TYPE "typeSmcChillerHrle90a40cmIo"
// stored: IsFailsafeCompliant false
   STRUCT
      in { ExternalAccessible := 'False'; ExternalVisible := 'False'; ExternalWritable := 'False'} : Struct   // Lesen / Read
         fluidDischargeTempCH1 { ExternalAccessible := 'False'; ExternalVisible := 'False'; ExternalWritable := 'False'} : Real;   // Austrittstemperatur der zirkulierenden Flüssigkeit Kanal 1 / Outlet temperature of the circulating fluid channel 1
         fluidDischargeTempCH2 { ExternalAccessible := 'False'; ExternalVisible := 'False'; ExternalWritable := 'False'} : Real;   // Austrittstemperatur der zirkulierenden Flüssigkeit Kanal 2 / Outlet temperature of the circulating fluid channel 2
         reserve1 { ExternalAccessible := 'False'; ExternalVisible := 'False'; ExternalWritable := 'False'} : Word;   // Reserve
         reserve2 { ExternalAccessible := 'False'; ExternalVisible := 'False'; ExternalWritable := 'False'} : Word;   // Reserve
         fluidDischargePressureCH1 { ExternalAccessible := 'False'; ExternalVisible := 'False'; ExternalWritable := 'False'} : Real;   // Förderdruck der zirkulierenden Flüssigkeit Kanal 1 / Delivery pressure of the circulating fluid channel 1
         reserve3 { ExternalAccessible := 'False'; ExternalVisible := 'False'; ExternalWritable := 'False'} : Word;   // Reserve
         reserve4 { ExternalAccessible := 'False'; ExternalVisible := 'False'; ExternalWritable := 'False'} : Word;   // Reserve
         reserve5 { ExternalAccessible := 'False'; ExternalVisible := 'False'; ExternalWritable := 'False'} : Word;   // Reserve
         dataDisplay1 { ExternalAccessible := 'False'; ExternalVisible := 'False'; ExternalWritable := 'False'} : Real;   // Datenanzeige 1 / Data display 1
         dataDisplay2 { ExternalAccessible := 'False'; ExternalVisible := 'False'; ExternalWritable := 'False'} : Real;   // Datenanzeige 2 / Data display 2
         statusFlags1 { ExternalAccessible := 'False'; ExternalVisible := 'False'; ExternalWritable := 'False'} : Array[0..15] of Bool;   // Statuskennzeichen 1 / Status identifier 1
         alarmFlags1 { ExternalAccessible := 'False'; ExternalVisible := 'False'; ExternalWritable := 'False'} : Array[0..15] of Bool;   // Alarmmerker 1 / Alarm flag 1
         alarmFlags2 { ExternalAccessible := 'False'; ExternalVisible := 'False'; ExternalWritable := 'False'} : Array[0..15] of Bool;   // Alarmmerker 2 / Alarm flag 2
         alarmFlags3 { ExternalAccessible := 'False'; ExternalVisible := 'False'; ExternalWritable := 'False'} : Array[0..15] of Bool;   // Alarmmerker 3 / Alarm flag 3
         alarmFlags4 { ExternalAccessible := 'False'; ExternalVisible := 'False'; ExternalWritable := 'False'} : Array[0..15] of Bool;   // Alarmmerker 4 / Alarm flag 4
         alarmFlags5 { ExternalAccessible := 'False'; ExternalVisible := 'False'; ExternalWritable := 'False'} : Array[0..15] of Bool;   // Alarmmerker 5 / Alarm flag 5
      END_STRUCT;
      inOut { ExternalAccessible := 'False'; ExternalVisible := 'False'; ExternalWritable := 'False'} : Struct   // Lesen/Schreiben / Read/write
         fluidSetTempCH1 { ExternalAccessible := 'False'; ExternalVisible := 'False'; ExternalWritable := 'False'} : Real;   // Solltemperatur der zirkulierenden Flüssigkeit / Target temperature of the circulating fluid
         fluidSetTempCH2 { ExternalAccessible := 'False'; ExternalVisible := 'False'; ExternalWritable := 'False'} : Real;   // Umwälzflüssigkeitssolltemperatur als Offset von Kanal 1 (Sollwert Kanal 2 = Sollwert Kanal 1 + Offset Kanal 2) / Circulating fluid target temperature as offset for channel 1 (target value channel 2 = target value channel 1 + offset channel 2)
         controlBits { ExternalAccessible := 'False'; ExternalVisible := 'False'; ExternalWritable := 'False'} : Array[0..15] of Bool;   // Steuerbits / Control bits
         dataInstr { ExternalAccessible := 'False'; ExternalVisible := 'False'; ExternalWritable := 'False'} : Array[0..1] of Byte;   // Datenanweisungen / Data instructions
      END_STRUCT;
   END_STRUCT;
   // // in.statusFlags1[0] : Laufstatus / Running status
   // // in.statusFlags1[1] : Betriebsstoppalarm ausgelöst Status / Stop operation alarm triggered status
   // // in.statusFlags1[2] : Betriebsfortsetzungsalarm ausgelöst / Continue operation alarm triggered
   // // in.statusFlags1[3] : Reserve
   // // in.statusFlags1[4] : Abschluss der Vorbereitung (TEMP READY) Status / End of preparation (TEMP READY) status
   // // in.statusFlags1[5] : Reserve
   // // in.statusFlags1[6] : Reserve
   // // in.statusFlags1[7] : Reserve
   // // in.statusFlags1[8] : Reserve
   // // in.statusFlags1[9] : Reserve
   // // in.statusFlags1[10] : Reserve
   // // in.statusFlags1[11] : Reserve
   // // in.statusFlags1[12] : Reserve
   // // in.statusFlags1[13] : Reserve
   // // in.statusFlags1[14] : Reserve
   // // in.statusFlags1[15] : Gefrierschutzstatus / Freeze protection status
   // // in.alarmFlags1[0] : Niedriger Flüssigkeitsstand im Tank / Low fluid level in the tank
   // // in.alarmFlags1[1] : CH1 abnorm hohe Temperatur der zirkulierenden Flüssigkeit / CH1 abnormally high temperature of the circulating fluid
   // // in.alarmFlags1[2] : Reserve
   // // in.alarmFlags1[3] : Reserve
   // // in.alarmFlags1[4] : Ungewöhnlich hohe Rücklauftemperatur der zirkulierenden Flüssigkeit / Unusually high return temperature of the circulating fluid
   // // in.alarmFlags1[5] : Ungewöhnlich hoher Auslassdruck der zirkulierenden Flüssigkeit / Unusually high outlet pressure of the circulating fluid
   // // in.alarmFlags1[6] : Reserve
   // // in.alarmFlags1[7] : Hoher Druckanstieg der zirkulierenden Flüssigkeit / High pressure increase of the circulating fluid
   // // in.alarmFlags1[8] : Hoher Druckabfall der zirkulierenden Flüssigkeit / High pressure of the circulating fluid
   // // in.alarmFlags1[9] : Reserve
   // // in.alarmFlags1[10] : Ungewöhnlich niedrige Ansaugtemperatur des Kompressors / Unusually low intake temperature of the compressor
   // // in.alarmFlags1[11] : Reserve
   // // in.alarmFlags1[12] : Unnormaler Anstieg des Drucks im Kältemittelkreislauf (Hochdruckseite) / Abnormal pressure rise in the coolant circuit (high pressure side)
   // // in.alarmFlags1[13] : Reserve
   // // in.alarmFlags1[14] : Kältemittelleck / Coolant leak
   // // in.alarmFlags1[15] : Ungewöhnlicher Anstieg des Drucks im Kältemittelkreislauf (Niederdrucksei / Unusual pressure rise in the coolant circuit (low pressure side)
   // // in.alarmFlags2[0] : Ungewöhnlicher Druckabfall im Kältemittelkreislauf (Niederdruckseite) / Unusual pressure drop in the coolant circuit (low pressure side)
   // // in.alarmFlags2[1] : Kompressor läuft nicht / Compressor not running
   // // in.alarmFlags2[2] : Kommunikationsfehler / Communication error
   // // in.alarmFlags2[3] : Reserve
   // // in.alarmFlags2[4] : Reserve
   // // in.alarmFlags2[5] : Ausfall des Temperatursensors für den Auslass der CH1-Umlaufflüssigkeit（PT1) / Failure of the temperature sensor for the outlet of the CH1 circulation fluid （PT1)
   // // in.alarmFlags2[6] : Ausfall des Rücklauftemperatursensors der zirkulierenden Flüssigkeit（PT2) / Failure of the circulating fluid return temperature sensor （PT2)
   // // in.alarmFlags2[7] : Verdichter-Saugtemperatursensor defekt（TH2) / Compressor intake temperature sensor defective（TH2)
   // // in.alarmFlags2[8] : Ausfall des Drucksensors für die zirkulierende Flüssigkeit （PS1） / Failure of the pressure sensor for the circulating fluid （PS1）
   // // in.alarmFlags2[9] : Drucksensor des Kältemittelkreislaufs (Hochdruckseite) defekt（PS2） / Pressure sensor of the coolant circuit (high pressure side) defective（PS2）
   // // in.alarmFlags2[10] : Drucksensor des Kältemittelkreislaufs (Niederdruckseite) defekt（PS3） / Pressure sensor of the coolant circuit (low pressure side) defective（PS3）
   // // in.alarmFlags2[11] : Reserve
   // // in.alarmFlags2[12] : Reserve
   // // in.alarmFlags2[13] : Reserve
   // // in.alarmFlags2[14] : Kontakteingang 1 Signalerkennung / Contact input 1 signal detection
   // // in.alarmFlags2[15] : Kontakteingang 2 Signalerkennung / Contact input 2 signal detection
   // // in.alarmFlags3[0] : Reserve
   // // in.alarmFlags3[1] : Anstieg der elektrischen Leitfähigkeit / Increase in electrical conductivity
   // // in.alarmFlags3[2] : Rückgang der elektrischen Leitfähigkeit / Decrease in electrical conductivity
   // // in.alarmFlags3[3] : Ausfall des elektrischen Leitfähigkeitssensors / Failure of the electrical conductivity sensor
   // // in.alarmFlags3[4] : Ausfall des Verdichter-Drucktemperatursensors （TH1) / Failure of the compressor pressure and temperature sensor （TH1)
   // // in.alarmFlags3[5] : Anstieg der Verdichter-Austrittstemperatur / Increase in compressor outlet temperature
   // // in.alarmFlags3[6] : Reserve
   // // in.alarmFlags3[7] : Reserve
   // // in.alarmFlags3[8] : Reserve
   // // in.alarmFlags3[9] : Reserve
   // // in.alarmFlags3[10] : Ausfall des Ventilators / Failure of the ventilator
   // // in.alarmFlags3[11] : Reserve
   // // in.alarmFlags3[12] : Reserve
   // // in.alarmFlags3[13] : Verdichter-Wechselrichter-Fehler / Compressor inverter error
   // // in.alarmFlags3[14] : Störung des Pumpenbetriebs / Pump operation fault
   // // in.alarmFlags3[15] : Fehler im Pumpenumrichter / Error in the pump inverter
   // // in.alarmFlags4[0] : Reserve
   // // in.alarmFlags4[1] : CH2 abnormal hohe Temperatur der zirkulierenden Flüssig / CH2 abnormally high temperature of the circulating fluid
   // // in.alarmFlags4[2] : Ausfall des Temperatursensors für den Auslass der CH2-Umlaufflüssigkeit（PT3） / Failure of the temperature sensor for the outlet of the CH2 circulation fluid （PT3)
   // // in.alarmFlags4[3] : Speicherfehler 1 / Storage error 1
   // // in.alarmFlags4[4] : Speicherfehler 2 / Storage error 2
   // // in.alarmFlags4[5] : Reserve
   // // in.alarmFlags4[6] : Reserve
   // // in.alarmFlags4[7] : Abnormale Missing-Phase / Anti-Phase / Abnormal missing phase / anti-phase
   // // in.alarmFlags4[8] : Kommunikationsfehler des Verdichterwechselrichters / Communication error of the compressor inverter
   // // in.alarmFlags4[9] : Parameterfehler des Pumpenumrichters / Pump inverter parameter error
   // // in.alarmFlags4[10] : Kommunikationsfehler des Pumpenumrichters / Communication error of the pump inverter
   // // in.alarmFlags4[11] : Hinweis zur Wartung / Note on preventive maintenance
   // // in.alarmFlags4[12] : Kommunikationsfehler / Communication error
   // // in.alarmFlags4[13] : Interner Kommunikationsfehler / Internal communication error
   // // in.alarmFlags4[14] : Druckanstieg im Kältemittelkreislauf (Hochdruckseite) / Pressure rise in the coolant circuit (high pressure side)
   // // in.alarmFlags4[15] : Fehler in der Stromversorgung / Error in the power supply
   // // in.alarmFlags5[0] : Schalterbetätigung für den Druck im Kältemittelkreislauf (Hochdruckseite) / Switch actuation for the pressure in the coolant circuit (high pressure side)
   // // in.alarmFlags5[1] : Parameterfehler des Verdichterumrichters / Compressor inverter parameter error
   // // in.alarmFlags5[2] : Reserve
   // // in.alarmFlags5[3] : Reserve
   // // in.alarmFlags5[4] : Reserve
   // // in.alarmFlags5[5] : Reserve
   // // in.alarmFlags5[6] : Reserve
   // // in.alarmFlags5[7] : Reserve
   // // in.alarmFlags5[8] : Reserve
   // // in.alarmFlags5[9] : Reserve
   // // in.alarmFlags5[10] : Reserve
   // // in.alarmFlags5[11] : Reserve
   // // in.alarmFlags5[12] : Reserve
   // // in.alarmFlags5[13] : Reserve
   // // in.alarmFlags5[14] : Reserve
   // // in.alarmFlags5[15] : Reserve
   // // inOut.controlBits[0] : Befehl zum Starten der Operation / Command for starting the operation
   // // inOut.controlBits[1] : Flagge für Modusanforderung / Flag for mode request
   // // inOut.controlBits[2] : Alarm-Reset-Flag / Alarm reset flag
   // // inOut.controlBits[3] : Reserve
   // // inOut.controlBits[4] : Reserve
   // // inOut.controlBits[5] : Reserve
   // // inOut.controlBits[6] : Reserve
   // // inOut.controlBits[7] : Reserve
   // // inOut.controlBits[8] : Reserve
   // // inOut.controlBits[9] : Reserve
   // // inOut.controlBits[10] : Reserve
   // // inOut.controlBits[11] : Reserve
   // // inOut.controlBits[12] : Reserve
   // // inOut.controlBits[13] : Reserve
   // // inOut.controlBits[14] : Reserve
   // // inOut.controlBits[15] : Reserve
   // // inOut.dataInstr[0] : Datenanweisung 1 / Data instruction 1
   // // inOut.dataInstr[1] : Datenanweisung 2 / Data instruction 2
END_TYPE

TYPE "typeSmcChillerHrle90a40cmStatus"
// stored: IsFailsafeCompliant false
   STRUCT
      fluidActualDischargeTempCh1 { ExternalAccessible := 'False'; ExternalVisible := 'False'; ExternalWritable := 'False'} : Real;   // Temperatur am Ausgang Kanal 1 / Temperature at the outlet channel 1
      fluidActualDischargeTempCh2 { ExternalAccessible := 'False'; ExternalVisible := 'False'; ExternalWritable := 'False'} : Real;   // Temperatur am Ausgang Kanal 2 / Temperature at the outlet channel 2
      fluidActualDischargePressureCh1 { ExternalAccessible := 'False'; ExternalVisible := 'False'; ExternalWritable := 'False'} : Real;   // Druck am Ausgang Kanal 1 / Pressure at the outlet channel 1
      fluidSetpointDischargeTempCh1 { ExternalAccessible := 'False'; ExternalVisible := 'False'; ExternalWritable := 'False'} : Real;   // Sollwert für die Flüssigkeitstemperatur Kanal 1 / Target value for the fluid temperature channel 1
      chillerRunning { ExternalAccessible := 'False'; ExternalVisible := 'False'; ExternalWritable := 'False'} : Bool;   // Kühlung läuft / Cooling running
      chillerInRemoteMode { ExternalAccessible := 'False'; ExternalVisible := 'False'; ExternalWritable := 'False'} : Bool;   // Kältemaschine im Remote-Modus / Cooling unit in Remote mode
      chillerTempReady { ExternalAccessible := 'False'; ExternalVisible := 'False'; ExternalWritable := 'False'} : Bool;   // Chiller-Prozessvorbereitung abgeschlossen / Chiller process preparation finished
      dataDisplay { ExternalAccessible := 'False'; ExternalVisible := 'False'; ExternalWritable := 'False'} : Struct   // Über die Datenanzeigeanweisung zurückgegebener Wert / Value returned via the data display instruction
         "1" { ExternalAccessible := 'False'; ExternalVisible := 'False'; ExternalWritable := 'False'} : Struct   // 1
            valueType { ExternalAccessible := 'False'; ExternalVisible := 'False'; ExternalWritable := 'False'} : Byte;   // Art des Wertes / Type of value
            value { ExternalAccessible := 'False'; ExternalVisible := 'False'; ExternalWritable := 'False'} : Real;   // Wert / Value
         END_STRUCT;
         "2" { ExternalAccessible := 'False'; ExternalVisible := 'False'; ExternalWritable := 'False'} : Struct   // 2
            valueType { ExternalAccessible := 'False'; ExternalVisible := 'False'; ExternalWritable := 'False'} : Byte;   // Art des Wertes / Type of value
            value { ExternalAccessible := 'False'; ExternalVisible := 'False'; ExternalWritable := 'False'} : Real;   // Wert / Value
         END_STRUCT;
      END_STRUCT;
      errorFB { ExternalAccessible := 'False'; ExternalVisible := 'False'; ExternalWritable := 'False'} : Struct   // Fehler im Funktionsblock / Error in the function block
         active { ExternalAccessible := 'False'; ExternalVisible := 'False'; ExternalWritable := 'False'} : Bool;   // Aktiv / Active
         errorLocation { ExternalAccessible := 'False'; ExternalVisible := 'False'; ExternalWritable := 'False'} : DWord;   // Ort des Fehlers / Error location
         errorCode { ExternalAccessible := 'False'; ExternalVisible := 'False'; ExternalWritable := 'False'} : DWord;   // Fehlercode / Error code
      END_STRUCT;
      alarmDevice { ExternalAccessible := 'False'; ExternalVisible := 'False'; ExternalWritable := 'False'} : Struct   // Alarm am Kühlgerät / Alarm at cooler
         active { ExternalAccessible := 'False'; ExternalVisible := 'False'; ExternalWritable := 'False'} : Bool;   // Aktiv / Active
      END_STRUCT;
      warningDevice { ExternalAccessible := 'False'; ExternalVisible := 'False'; ExternalWritable := 'False'} : Struct   // Warnung am Kühlgerät / Warning on the cooling unit
         active { ExternalAccessible := 'False'; ExternalVisible := 'False'; ExternalWritable := 'False'} : Bool;   // Aktiv / Active
      END_STRUCT;
   END_STRUCT;
END_TYPE

TYPE "typeMotion"
TITLE = Movement / Bewegung
// Movement [V 01.00 | Kernel_V2] / Bewegung [V 01.00 | Kernel_V2]
// stored: IsFailsafeCompliant false
   STRUCT
      autoToPos : Bool;   // Automatic to Position / Automatic to position
      inPosition : Bool;   // In Position / In position
      autoInPos : Bool;   // In Position Automatic / In position automatic
      toPosition : Bool;   // To Position
   END_STRUCT;
END_TYPE

TYPE "typeGroupOvrvList"
TITLE = Overview of groups / Gruppenübersicht
// Group overview [V 01.00 | Kernel_V2] / Gruppenübersicht [V 01.00 | Kernel_V2]
// stored: IsFailsafeCompliant false
   STRUCT
      lastUsedIndex : DInt := -1;   // Letzter Benutzter Index / Last user index
      valid : Bool;   // Gültigkeit / Scope
      overflowCount : DInt;   // Gruppen Überlauf Zähler / Groups overtravel counter
      firstListedCortArea : DInt := -1;   // Index der ersten gelisteten CA / Index of first listed CA
      groups : Array[0.."MAX_CNT_GRP_OVR_ENTRIES"] of "typeGroupOvrvListEntry";   // Gruppen (CAs/CGs/FGs) / Groups (CAs/CGs/FGs)
   END_STRUCT;
END_TYPE

TYPE "typeGroupOvrvListEntry"
TITLE = Entry group overview / Eintrag Gruppenübersicht
// Entry group overview [V 01.00 | Kernel_V2] / Eintrag Gruppenübersicht [V 01.00 | Kernel_V2]
// stored: IsFailsafeCompliant false
   STRUCT
      alive : USInt;   // Alive-Flag (Wird in der Gruppe gesetzt, zentral dann zurückgesetzt) / Alive-Flag (is set in group, then centrally reset)
      dbAnyAddr : DB_ANY;   // DB-Any Adresse (typeCaCgFg) / DB any address (typeCaCgFg)
      nextPartnerIndex : DInt := -1;   // Index der Nächsten Partner-Gruppe / Index of next partner group
      firstChildIndex : DInt := -1;   // Index der ersten untergeordneten Gruppe / Index of first subordinate group
   END_STRUCT;
END_TYPE

TYPE "typeFaultManagement"
TITLE = Error management / Fehlerverwaltung
// Fehlerverwaltung [V 01.01 | Kernel_V2]
// stored: IsFailsafeCompliant false
   STRUCT
      selectAckFault : Bool;   // Anwahl Störung quittieren (S) / Selection: acknowledge fault (S)
      ackFault : Bool;   // Störung quittieren / Acknowledge fault
      faultGeneral : Bool;   // Generelle Störung steht an / General fault pending
      faultInstantStop : Bool;   // Störung sofort Halt steht an / Fault immediate stop pending
      faultMachineOut : Bool;   // Störung sofort Halt und Maschine Aus steht an / Fault immediate stop and machine off pending
      faultInCycleEnd : Bool;   // Störung Halt nach Taktende steht an / Fault stop at end of cycle pending
      faultNoStop : Bool;   // Störung ohne Stop steht an / Fault without stop pending
      faultActive : Bool;   // Störung ist aktiv (aus eigener oder übergeordeten Gruppen) / Fault is active (from separate or superordinate groups)
      messageGeneral : Bool;   // Meldung steht an / Message pending
      messageOperatorCall : Bool;   // Meldung mit Bedienerruf steht an / Message with operator call pending
      selectInstantStop : Bool;   // Anwahl sofort Halt bei Störung (S) / Selection immediate stop in case of fault (S)
      selectMachineOut : Bool;   // Anwahl sofort Halt und Maschine aus (S)
      selectStopCycleEnd : Bool;   // Anwahl Halt nach Taktende bei Störung (S) / Selection stop at end of cycle in case of fault (S)
      faultInstantStopByParent : Bool;   // Störung sofort Halt von übergeordneter Baugruppe / Fault immediate stop from superordinate assembly
      faultInCycleEndByParent : Bool;   // Störung Halt nach Taktende von übergeordneter Baugruppe / Fault stop at end of cycle from the superordinate assembly
   END_STRUCT;
END_TYPE

TYPE "typeProDiagEvaluation"
TITLE = ProDiag evaluation / ProDiag Auswertung
// ProDiag evaluation [V 01.00 | Kernel_V2] / ProDiag Auswertung [V 01.00 | Kernel_V2]
// stored: IsFailsafeCompliant false
   STRUCT
      faultInstantStop : Bool;   // Störung sofort Halt steht an / Fault immediate stop pending
      faultNoStop : Bool;   // Störung ohne Stop steht an / Fault without stop pending
      faultInCycleEnd : Bool;   // Störung Halt nach Taktende steht an / Fault stop at end of cycle pending
      faultMachineOut : Bool;   // Störung sofort Halt und Maschine Aus steht an / Fault immediate stop and machine off pending
      faultSequence : Bool;   // Ablaufstörung steht an / Sequence fault pending
      message : Bool;   // Meldung steht an / Message pending
      messageOperatorCall : Bool;   // Meldung mit Bedienerruf steht an / Message with operator call pending
      information : Bool;   // Information steht an / Information pending
      popUp : Bool;   // PopUp steht an / Popup pending
      criteriaAnalysis : Bool;   // Kriterienanalyse steht an / Criteria analysis pending
      plcCodeDisplay : Bool;   // Plc Code Anzeige steht an / PLC code display pending
   END_STRUCT;
END_TYPE

TYPE "typeSbtData"
TITLE = typeSbtData
// stored: IsFailsafeCompliant false
   STRUCT
      BrakeTestRequest { ExternalAccessible := 'False'; ExternalVisible := 'False'; ExternalWritable := 'False'} : Bool := false;   // Bremsentest Anforderung
      BrakeTestRequestWithPreconditions { ExternalAccessible := 'False'; ExternalVisible := 'False'; ExternalWritable := 'False'} : Bool := false;   // Bremsentest Anforderung mit Vorbedingungen
      BrakeTestPreconditionsNOK { ExternalAccessible := 'False'; ExternalVisible := 'False'; ExternalWritable := 'False'} : Bool := false;   // Bremsentest Vorbedingungen NOK
      BrakeTestImmediately { ExternalAccessible := 'False'; ExternalVisible := 'False'; ExternalWritable := 'False'} : Bool := false;   // Sofortausführung Bremsentest
      BrakeTestActive { ExternalAccessible := 'False'; ExternalVisible := 'False'; ExternalWritable := 'False'} : Bool := false;   // Bremsentest ist zur Zeit aktiv
      SafeGuardBlocked { ExternalAccessible := 'False'; ExternalVisible := 'False'; ExternalWritable := 'False'} : Bool := false;   // Öffnen/Entriegeln der Schutzteinrichtung ist geblockt
   END_STRUCT;
END_TYPE

TYPE "typeTeststoppSBTData"
// V 01.00
// stored: IsFailsafeCompliant false
   STRUCT
      BrakeTestRequest { S7_SetPoint := 'True'} : Bool := false;   // Bremsentest Anforderung / Brake test request
      BrakeTestRequestWithPreconditions : Bool;   // Bremsentest Anforderung mit Vorbedingungen / Brake test request with preconditions
      BrakeTestPreconditionsNOK : Bool;   // Bremsentest Vorbedingungen NOK / Brake test preconditions NOK
      BrakeTestImmediately { S7_SetPoint := 'True'} : Bool := false;   // Sofortausführung Bremsentest / Immediate execution brake test
      BrakeTestActive : Bool;   // Bremsentest ist zur Zeit aktiv / Brake test is currently active
      SafeGuardBlocked { S7_SetPoint := 'True'} : Bool := false;   // Öffnen/Entriegeln der Schutzteinrichtung ist geblockt / Opening/unlocking the safeguard is blocked
   END_STRUCT;
END_TYPE

TYPE "typeTeststoppSBTError"
// V 01.00
// stored: IsFailsafeCompliant false
   STRUCT
      BrakeTestParameter { S7_SetPoint := 'True'} : Bool := false;   // Störung: Bremsentest-Parameter / Fault: brake test parameter
      BrakeTestSequenceFault : Bool;   // Störung: Ablaufstörung Teststopp/Bremsentest / Fault: sequence fault test stop/brake test
      BrakeTestIntBrake : Bool;   // Störung: Bremsentest interne Bremse fehlgeschlagen / Fault: brake test internal brake failed
      BrakeTestExtBrake : Bool;   // Störung: Bremsentest externe Bremse fehlgeschlagen / Fault: brake test external brake failed
   END_STRUCT;
END_TYPE

TYPE "typeTeststoppSBTPopUpWarn"
// V 01.00
// stored: IsFailsafeCompliant false
   STRUCT
      DoNotOpenSafeGuard : Bool;   // Bremsentest/Teststopp aktiv => Schutzeinrichtung nicht unterbrechen/öffnen / Brake test/test stop active => do not interrupt/open safeguard
      SafeGuardNotOpen { S7_SetPoint := 'True'} : Bool := false;   // Bremsentest/Teststopp angefordert => Schutzeinrichtung kann nicht geöffnet/entriegelt werden (Leistung ein oder E2 erforderlich) / Brake test/test stop requested => safeguard cannot be opened/unlocked (power on or E2 required)
      BrakeTestImmediately { S7_SetPoint := 'True'} : Bool := false;   // Schutzeinrichtung für Bremsentest/Teststopp schließen oder quittieren / Close or acknowledge safeguard for brake test/test stop
      BrakeTestNioPowerOff { S7_SetPoint := 'True'} : Bool := false;   // Bremsentest nio => Leistung aus (Bremse/Antrieb austauschen) / Brake test NOK => power off (exchange brake/drive)
      BrakeTestOnlyInHome : Bool;   // Bremsentest/Teststopp ist nur in Grundstellung möglich / Brake test/test stop only possible in home position
   END_STRUCT;
END_TYPE

TYPE "typeTeststoppSbtSummary"
TITLE = typeTeststoppSbtSummary
// stored: IsFailsafeCompliant false
   STRUCT
      safeGuardBlockedCollectSafeArea { ExternalAccessible := 'False'; ExternalVisible := 'False'; ExternalWritable := 'False'} : Bool := false;   // Öffnen/Entriegeln der Schutzeinrichtung ist geblockt
      brakeTestActiveCollectSafeArea { ExternalAccessible := 'False'; ExternalVisible := 'False'; ExternalWritable := 'False'} : Bool := false;   // Bremsentest ist aktiv
      brakeTestNioCollected { ExternalAccessible := 'False'; ExternalVisible := 'False'; ExternalWritable := 'False'} : Bool := false;   // Bremsentest nio gesammelt
   END_STRUCT;
END_TYPE

TYPE "API_Inputs"
// stored: IsFailsafeCompliant false
   STRUCT
      Heartbeat : Bool;   // Heartbeat Input from Middleware
      Ready : Bool;   // Middleware Ready for Transations
      Job_Comp : Bool;   // Middleware Job has Been Completed
      Clear_Results : Bool;   // Clear Results Stored in PLC. Set by Middleware
      Mutex : Bool;   // Mutex Token with Middleware to Prevent Multiple Instances Running
      Rx : DInt;   // Recieved Counter
      Active_Job : DInt;   // Current Job Active in Middleware
      Fault_Code : Array[0..9] of DInt;   // Fault Code from Middleware
      Timeout : Time;   // Timeout Value for SIS Job. Value set by Middleware and is dependant upon Job Function.
      LDD : Struct   // Laser Depth Dynamics
         Ref_Plane : DInt;
         Status : Struct   // Current Status of the LDD System (Pseudo DIO)
            OK : Bool;   // LDD System is OK
            Ready_Cmd : Bool;   // LDD System is Ready to Recieve a Command
            Wait_Trigger : Bool;   // LDD System is Waiting for Trigger
            Acquiring : Bool;   // LDD System is Acquiring Data
            Remote_Control : Bool;   // LDD is in Remote Mode
            Seq_Complete : Bool;   // Overall Sequence is Complete
            Seq_Pass : Bool;   // Overall Sequence has Passed
            Seq_Fail : Bool;   // Overall Sequence has Failed
         END_STRUCT;
         DDO : Array[0.."LASERCOMM_LDD_ARRAY_SIZE"] of "LaserComm_DDO";   // Array for Storage of Measurement Data from LDD
         Results : Array[0.."LASERCOMM_LDD_ARRAY_SIZE"] of "LaserComm_LDD_Results";   // Array for Storage of LDD QA Results
      END_STRUCT;
      YLR { S7_SetPoint := 'True'} : "YLR_Inputs";   // Inputs from YLR Laser (signals handled by Middleware)
   END_STRUCT;
END_TYPE

TYPE "API_Outputs"
// stored: IsFailsafeCompliant false
   STRUCT
      Job_Comp_Ack : Bool;   // Acknowledge the Job Complete Signal has been Received
      Tx : DInt;   // Transmission Counter
      Job : DInt;   // Middleware Job Command
      Serial_Number : Array[1..32] of Char;   // Serial Number of Part to Be Loaded to LDD File
      Part_Type : Array[1..18] of Char;   // Part Type in Station
      LDD : Struct   // Laser Depth Dynamics
         Sequence_Mask : Array[0.."LASERCOMM_LDD_ARRAY_SIZE"] of Bool;   // Weld Mask for Skipping Welds in an LDD Sequence
      END_STRUCT;
   END_STRUCT;
END_TYPE

TYPE "API_Parameters"
// stored: IsFailsafeCompliant false
   STRUCT
      Placeholder : Bool;   // No Parameters Required as of update. Placeholder Tag as accurate offsetting is required.
   END_STRUCT;
END_TYPE

TYPE "LaserComm_DDO"
// stored: IsFailsafeCompliant false
   STRUCT
      Valid : Bool;   // Data Loaded from Laser Comm and is Valid
      Min : Real;   // Minimum Point Value from LDD Measurement
      Max : Real;   // Maximum Point Value from LDD Measurement
      Mean : Real;   // Average Point Value from LDD Measurement
      Dev : Real;   // Standard Deviation of LDD Measurement
   END_STRUCT;
END_TYPE

TYPE "LaserComm_Instance"
// stored: IsFailsafeCompliant false
   STRUCT
      API : Struct   // Tags associated with JLR Middleware and LDD
         Job : DInt;   // API Job - Triggers Job to Middleware. Value Clears on Completion of Job
         Faults : DInt;   // Faults Generated from SIS Interface. Set Bitwise
         Reset : Bool;   // Reset API
         Inputs : "API_Inputs";   // Inputs to API. Set from Middleware
         Outputs { S7_SetPoint := 'True'} : "API_Outputs";   // Outputs from API. Read by Middleware
         Parameters { S7_SetPoint := 'True'} : "API_Parameters";   // API Parameters
      END_STRUCT;
      Scanner : Struct   // Tags associated with IPG Scanner Software and Hardware
         oJob : Byte;   // Output Job Number to IPG Weld
         oGroup : Byte;   // Output Group Number to IPG Weld
         iJob : Byte;   // Input Running Job Number from IPG
         iGroup : Byte;   // Input Running Group Number from IPG Weld
         Faults : DInt;   // Faults Generated from IPG Interface. Set Bitwise
         Start : Bool;   // Start Command to IPG Weld to Execute Weld Job
         Waiting_Start : Bool;   // IPG Weld is Waiting for a Start Signal. Job and Group have been Loaded
         Waiting_Strobe : Bool;   // IPG Weld is Ready for a New Job and Group Load
         Reset : Bool;   // Reset IPG Weld Interface
         Weld_Offset : Struct   // Offset Values of Weld Position. Can be expanded to array. Not support at present.
            X : Real;   // X
            Y : Real;   // Y
            Z : Real;   // Z
            "A" : Real;   // A
            "B" : Real;   // B
            C : Real;   // C
         END_STRUCT;
      END_STRUCT;
      Static : Struct   // Static Tags used internally to Laser Comm FBs
         IPG_Job_Complete : Bool;   // IPG Weld Job has Completed
         LDD_Job_Loaded : Bool;   // LDD Sequence has been Loaded for the Part
         OverPen_Detected : Bool;   // LDD has Reported an Over Penetration. Flag set in FB.
      END_STRUCT;
   END_STRUCT;
END_TYPE

TYPE "LaserComm_LDD_Results"
// stored: IsFailsafeCompliant false
   STRUCT
      QA : DInt;   // Pass/Fail for the LDD Job (0= Incomplete, 1=Pass, 2= Fail, 3=No QA)
      Warning : DInt;   // Warning Code for the LDD Job (0= Incomplete, 1=Pass, 2= Fail, 3=No QA)
      Reasons : Struct   // Reason for Weld QA Failure
         KHD : DInt;   // Keyhole Depth Measurement
         FWS : DInt;   // Finished Weld Surface Measurement
         XSP : DInt;   // Cross Section Parameter Measurement
         SPO : DInt;   // Seam Position Measurement
         SLE : DInt;   // Seam Left Edge Measurement
         SRE : DInt;   // Seam Right Edge Measurement
         SLH : DInt;   // Seam Left Height Measurement
         SRH : DInt;   // Seam Right Height Measurement
         SHH : DInt;   // Seam Step Height Measurement
         SCP : DInt;   // Seam Centre Position Measurement
         SGP : DInt;   // Seam Gap Width Measurement
         SJP : DInt;   // Seam Joint Feature Position Measurement
         SJH : DInt;   // Seam Joint Feature Height Measurement
         WPH : DInt;   // Workpiece Height Measurement
         TLE : DInt;   // Transverse Profile Left Edge Position Measurement
         TRE : DInt;   // Transverse Profile Right Edge Position Measurement
         TBD : DInt;   // Weld Bead Centre Measurement
         TBW : DInt;   // Weld Bead Width Measurement
      END_STRUCT;
   END_STRUCT;
END_TYPE

TYPE "Scanner_Inputs"
// stored: IsFailsafeCompliant false
   STRUCT
      Ready : Bool;   // Ready
      Active : Bool;   // Active
      Error : Bool;   // Error
      Status_Reserved : Bool;   // Status_Reserved
      DefinitionID_0 : Bool;   // DefinitionID_0
      DefinitionID_1 : Bool;   // DefinitionID_1
      DefinitionID_2 : Bool;   // DefinitionID_2
      DefinitionID_3 : Bool;   // DefinitionID_3
      Software_Status_Code { S7_SetPoint := 'True'} : Byte;   // Software_Status_Code
      Software_Status_Bit : Byte;   // Software_Status_Bit
      Status_Reserved_1 : Byte;   // Status_Reserved_1
      GPO_0 : Bool;   // GPO_0
      GPO_1 : Bool;   // GPO_1
      GPO_2 : Bool;   // GPO_2
      GPO_3 : Bool;   // GPO_3
      GPO_4 : Bool;   // GPO_4
      GPO_5 : Bool;   // GPO_5
      GPO_6 : Bool;   // GPO_6
      GPO_7 : Bool;   // GPO_7
      GPO_8 : Bool;   // GPO_8
      GPO_9 : Bool;   // GPO_9
      GPO_10 : Bool;   // GPO_10
      GPO_11 : Bool;   // GPO_11
      "Port_C Reserved_0" : Bool;   // Port_C Reserved_0
      "Port_C Reserved_1" : Bool;   // Port_C Reserved_1
      "Port_C Reserved_2" : Bool;   // Port_C Reserved_2
      "Port_C Reserved_3" : Bool;   // Port_C Reserved_3
      Group_ID_Feedback { S7_SetPoint := 'True'} : Byte;   // Group_ID_Feedback
      Job_ID_Feedback : Byte;   // Job_ID_Feedback
      Aborting : Bool;   // Aborting
      FIFO_Underrun : Bool;   // FIFO_Underrun
      Status_2_Reserved : Bool;   // Status_2_Reserved
      Hardware_Error : Bool;   // Hardware_Error
      Controller_Communication_Not_Detected : Bool;   // Controller_Communication_Not_Detected
      Controller_Communication_Error : Bool;   // Controller_Communication_Error
      Head_Communication_Not_Detected : Bool;   // Head_Communication_Not_Detected
      Head_Communication_Error : Bool;   // Head_Communication_Error
      XY_Hardware_Error : Bool;   // XY_Hardware_Error
      Z_Hardware_Error : Bool;   // Z_Hardware_Error
      XY_Position_Error : Bool;   // XY_Position_Error
      Z_Position_Error : Bool;   // Z_Position_Error
      Status_2_Reserved_1 : Bool;   // Status_2_Reserved_1
      Beam_Blocked : Bool;   // Beam_Blocked
      Tray_Missing : Bool;   // Tray_Missing
      Fibre_Interlock_Error : Bool;   // Fibre_Interlock_Error
      "Laser_Alarm_0/Ready" : Bool;   // Laser_Alarm_0/Ready
      "Laser_Alarm_1/Error" : Bool;   // Laser_Alarm_1/Error
      "Laser_Alarm_2/Emission_On" : Bool;   // Laser_Alarm_2/Emission_On
      "Laser_Alarm_3/Airflow" : Bool;   // Laser_Alarm_3/Airflow
      Laser_Not_Ready : Bool;   // Laser_Not_Ready
      Sync_Unlocked : Bool;   // Sync_Unlocked
      Status_2_Reserved_2 : Bool;   // Status_2_Reserved_2
      Status_2_Reserved_3 : Bool;   // Status_2_Reserved_3
      Stage_A_Error : Bool;   // Stage_A_Error
      Stage_B_Error : Bool;   // Stage_B_Error
      Stage_C_Error : Bool;   // Stage_C_Error
      Stage_D_Error : Bool;   // Stage_D_Error
      Clipping : Bool;   // Clipping
      Status_2_Reserved_4 : Bool;   // Status_2_Reserved_4
      Status_2_Reserved_5 : Bool;   // Status_2_Reserved_5
      Status_2_Reserved_6 : Bool;   // Status_2_Reserved_6
      Protective_Window_Photodiode_Feedback : Int;   // Protective_Window_Photodiode_Feedback
      Head_Temperature : Word;   // Head_Temperature
      Laser_Enable : Bool;   // Laser_Enable
      Laser_Gate : Bool;   // Laser_Gate
      Primary_Laser_Modulation : Bool;   // Primary_Laser_Modulation
      Guide_Laser : Bool;   // Guide_Laser
      Focus_Enable : Bool;   // Focus_Enable
      Port_B_Reserved : Bool;   // Port_B_Reserved
      Port_B_Reserved_1 : Bool;   // Port_B_Reserved_1
      Port_B_Reserved_2 : Bool;   // Port_B_Reserved_2
      Commanded_Core_Laser_Power : Byte;   // Commanded_Core_Laser_Power
      Port_B_Reserved_3 : Byte;   // Port_B_Reserved_3
      Commanded_Ring_Laser_Power : Byte;   // Commanded_Ring_Laser_Power
      Finished_Frame_ID : DInt;   // Finished_Frame_ID
      Finished_Object_ID : DInt;   // Finished_Object_ID
      Finished_Group_ID : DInt;   // Finished_Group_ID
      Frames_in_FIFO : DInt;   // Frames_in_FIFO
      Objects_in_FIFO : Int;   // Objects_in_FIFO
      Groups_in_FIFO : Int;   // Groups_in_FIFO
      XY_Position : Bool;   // XY_Position
      "Timer/Counter" : Bool;   // Timer/Counter
      Start : Bool;   // Start
      Wait_Status_Reserved : Bool;   // Wait_Status_Reserved
      Laser_Ready : Bool;   // Laser_Ready
      Interlock_OK : Bool;   // Interlock_OK
      Software_Wait : Bool;   // Software_Wait
      Group_Committed : Bool;   // Group_Committed
      GPI_0 : Bool;   // GPI_0
      GPI_1 : Bool;   // GPI_1
      GPI_2 : Bool;   // GPI_2
      GPI_3 : Bool;   // GPI_3
      Wait_Status_Reserved_1 : Bool;   // Wait_Status_Reserved_1
      Wait_Status_Reserved_2 : Bool;   // Wait_Status_Reserved_2
      Wait_Status_Reserved_3 : Bool;   // Wait_Status_Reserved_3
      Wait_Status_Reserved_4 : Bool;   // Wait_Status_Reserved_4
      In_View_X { S7_SetPoint := 'True'} : Bool;   // In_View_X
      In_View_Y : Bool;   // In_View_Y
      In_View_Z : Bool;   // In_View_Z
      Coordinate_Change_Done : Bool;   // Coordinate_Change_Done
      Encoder_Reset_A : Bool;   // Encoder_Reset_A
      Encoder_Reset_B : Bool;   // Encoder_Reset_B
      Encoder_Reset_C : Bool;   // Encoder_Reset_C
      Wait_Status_Reserved_5 : Bool;   // Wait_Status_Reserved_5
      Move_Done_A : Bool;   // Move_Done_A
      Move_Done_B : Bool;   // Move_Done_B
      Move_Done_C : Bool;   // Move_Done_C
      Wait_Status_Reserved_6 : Bool;   // Wait_Status_Reserved_6
      Wait_Status_Reserved_7 : Bool;   // Wait_Status_Reserved_7
      Wait_Status_Reserved_8 : Bool;   // Wait_Status_Reserved_8
      Wait_Status_Reserved_9 : Bool;   // Wait_Status_Reserved_9
      Wait_Status_Reserved_10 : Bool;   // Wait_Status_Reserved_10
   END_STRUCT;
END_TYPE

TYPE "Scanner_Outputs"
// stored: IsFailsafeCompliant false
   STRUCT
      Start : Bool;   // Command to Start IPG Weld Job
      Enable : Bool;   // Enable Scanner (Always On)
      Control_Reserved : Bool;
      Control_Reserved_1 : Bool;
      Control_Reserved_2 : Bool;
      Control_Reserved_3 : Bool;
      Control_Reserved_4 : Bool;
      Control_Reserved_5 : Bool;
      Control_Reserved_6 { S7_SetPoint := 'True'} : Byte;
      Control_Reserved_7 : Int;
      "GPI_0/Strobe" : Bool;   // Strobe for IPG Weld to Load a New Job
      GPI_1 : Bool;
      GPI_2 : Bool;
      GPI_3 : Bool;
      GPI_4 : Bool;
      GPI_5 : Bool;
      GPI_6 : Bool;
      GPI_7 : Bool;
      GPI_8 : Bool;
      GPI_9 : Bool;
      GPI_10 : Bool;
      GPI_11 : Bool;
      GPI_12 : Bool;
      GPI_13 : Bool;
      GPI_14 : Bool;
      GPI_15 : Bool;
      Group_ID_Select : Byte;   // Group to be Loaded
      Job_ID_Select : Byte;   // Job to Be Loaded
      Register_A : DInt;
      Register_B : DInt;
      Register_C : DInt;
   END_STRUCT;
END_TYPE

TYPE "YLR_Inputs"
// stored: IsFailsafeCompliant false
   STRUCT
      Command_Buffer_Overflow : Bool;   // Command_Buffer_Overflow
      Overheat : Bool;   // Overheat
      Emission_On : Bool;   // Emission_On
      High_Back_Reflection : Bool;   // High_Back_Reflection
      Analogue_Power_Control_Enabled : Bool;   // Analogue_Power_Control_Enabled
      Pulse_Too_Long : Bool;   // Pulse_Too_Long
      Reserved_1 : Bool;   // Reserved_1
      Reserved_2 : Bool;   // Reserved_2
      Aiming_Beam_On : Bool;   // Aiming_Beam_On
      Pulse_Too_Short : Bool;   // Pulse_Too_Short
      Pulsed_Mode : Bool;   // Pulsed_Mode
      Power_Supply_Off : Bool;   // Power_Supply_Off
      Modulation_Enabled : Bool;   // Modulation_Enabled
      Reserved_3 : Bool;   // Reserved_3
      Reserved_4 : Bool;   // Reserved_4
      Emission_Starting : Bool;   // Emission_Starting
      Gate_Mode_Enabled : Bool;   // Gate_Mode_Enabled
      High_Pulse_Energy : Bool;   // High_Pulse_Energy
      Hardware_Emission_Control_Enabled : Bool;   // Hardware_Emission_Control_Enabled
      Power_Supply_Failure : Bool;   // Power_Supply_Failure
      Front_Panel_Display_Locked : Bool;   // Front_Panel_Display_Locked
      Keyswitch_in_REM_Position : Bool;   // Keyswitch_in_REM_Position
      Waveform_Mode_On : Bool;   // Waveform_Mode_On
      Duty_Cycle_Too_High : Bool;   // Duty_Cycle_Too_High
      Low_Temperature : Bool;   // Low_Temperature
      Power_Supply_Alarm : Bool;   // Power_Supply_Alarm
      Reserved_5 : Bool;   // Reserved_5
      Hardware_Aiming_Beam_Control_Enabled : Bool;   // Hardware_Aiming_Beam_Control_Enabled
      Aiming_Beam_Alarm : Bool;   // Aiming_Beam_Alarm
      Critical_Error : Bool;   // Critical_Error
      Fiberlock_Interlock_Active : Bool;   // Fiberlock_Interlock_Active
      High_Average_Power : Bool;   // High_Average_Power
   END_STRUCT;
END_TYPE

TYPE "YLS_Inputs"
// stored: IsFailsafeCompliant false
   STRUCT
      Laser_Assigned : Bool;   // Laser_Assigned
      Laser_On : Bool;   // Laser_On
      System_Error : Bool;   // System_Error
      Guide_Laser_On : Bool;   // Guide_Laser_On
      Program_Active : Bool;   // Program_Active
      End_of_Program : Bool;   // End_of_Program
      Program_Interrupted : Bool;   // Program_Interrupted
      Analogue_Control_On : Bool;   // Analogue_Control_On
      System_Warning : Bool;   // System_Warning
      Laser_Ready : Bool;   // Laser_Ready
      Emission_On : Bool;   // Emission_On
      Synchronization_Output : Bool;   // Synchronization_Output
      Robot_Mode : Bool;   // Robot_Mode
      Power_Supply_Interlock : Bool;   // Power_Supply_Interlock
      Laser_Enabled : Bool;   // Laser_Enabled
      LaserNet_Control : Bool;   // LaserNet_Control
      Output_Power : Int;   // Output_Power
      Optical_Channel : Byte;   // Optical_Channel
      Program_Number : Byte;   // Program_Number
      Laser_Error : Bool;   // Laser_Error
      Laser_Warning : Bool;   // Laser_Warning
      Chiller_Error : Bool;   // Chiller_Error
      Chiller_Warning : Bool;   // Chiller_Warning
      Safety_Interlock_Open : Bool;   // Safety_Interlock_Open
      Channel_Error : Bool;   // Channel_Error
      Laser_Busy : Bool;   // Laser_Busy
      Slot_Error : Bool;   // Slot_Error
      Cabinet_Door_Open : Bool;   // Cabinet_Door_Open
      Reserved_Option_On : Bool;   // Reserved_Option_On
      Reduced_Output_Power : Bool;   // Reduced_Output_Power
      High_Back_Reflection : Bool;   // High_Back_Reflection
      Module_Without_Voltage_Supply : Bool;   // Module_Without_Voltage_Supply
      Piercing_Mode : Bool;   // Piercing_Mode
      Single_Module_Mode : Bool;   // Single_Module_Mode
      Reserved : Bool;   // Reserved
      Laser_Number : Byte;   // Laser_Number
      Reserved_1 : Byte;   // Reserved_1
      Modules_Selection : Int;   // Modules_Selection
      Core_Modules_Actual_Power : Int;   // Core_Modules_Actual_Power
      Ring_Modules_Actual_Power : Int;   // Ring_Modules_Actual_Power
   END_STRUCT;
END_TYPE

TYPE "YLS_Outputs"
// stored: IsFailsafeCompliant false
   STRUCT
      Laser_Request : Bool;   // Laser_Request
      Laser_On : Bool;   // Laser_On
      Reset_Errors : Bool;   // Reset_Errors
      Guide_Laser_On : Bool;   // Guide_Laser_On
      Program_Start : Bool;   // Program_Start
      Program_Stop : Bool;   // Program_Stop
      Reserved : Bool;   // Reserved
      Analogue_Control_On : Bool;   // Analogue_Control_On
      Control_by_LaserNet : Bool;   // Control_by_LaserNet
      Set_Rise_Time : Bool;   // Set_Rise_Time
      Set_Fall_Time : Bool;   // Set_Fall_Time
      Synchronization_Input : Bool;   // Synchronization_Input
      Reserved_1 : Bool;   // Reserved_1
      Piercing_Mode : Bool;   // Piercing_Mode
      Single_Module_Mode : Bool;   // Single_Module_Mode
      External_Error : Bool;   // External_Error
      Power : Int;   // Power
      Optical_Channel : Byte;   // Optical_Channel
      Program_Number : Byte;   // Program_Number
      Ramping_Time : Int;   // Ramping_Time
      Laser_Number : Byte;   // Laser_Number
      Reserved_2 : Byte;   // Reserved_2
      Modules_Selection : Int;   // Modules_Selection
      Core_Modules_Power_Setpoint : Int;   // Core_Modules_Power_Setpoint
      Ring_Modules_Power_Setpoint : Int;   // Ring_Modules_Power_Setpoint
   END_STRUCT;
END_TYPE

TYPE "typeKeyenceDetailedQuality"
// 01.00
// stored: IsFailsafeCompliant false
   STRUCT
      overall { ExternalAccessible := 'False'; ExternalVisible := 'False'; ExternalWritable := 'False'} : Char;   // Gesamtgüte / Overall quality
      overall_comma { ExternalAccessible := 'False'; ExternalVisible := 'False'; ExternalWritable := 'False'} : Char := ',';   // Komma / Comma
      dec { ExternalAccessible := 'False'; ExternalVisible := 'False'; ExternalWritable := 'False'} : Char;   // Deokdierung erfolgreich / fehlgeschlagen / Decoding successful / failed
      dec_comma { ExternalAccessible := 'False'; ExternalVisible := 'False'; ExternalWritable := 'False'} : Char := ',';   // Komma / Comma
      cc { ExternalAccessible := 'False'; ExternalVisible := 'False'; ExternalWritable := 'False'} : Char;   // Zellenkontrast / Cell contrast
      cc_comma { ExternalAccessible := 'False'; ExternalVisible := 'False'; ExternalWritable := 'False'} : Char := ',';   // Komma / Comma
      ccValue1 { ExternalAccessible := 'False'; ExternalVisible := 'False'; ExternalWritable := 'False'} : Char;   // Zellenkontrast (Wert) / Cell contrast (value)
      ccValue2 { ExternalAccessible := 'False'; ExternalVisible := 'False'; ExternalWritable := 'False'} : Char;   // Zellenkontrast (Wert) / Cell contrast (value)
      ccValue3 { ExternalAccessible := 'False'; ExternalVisible := 'False'; ExternalWritable := 'False'} : Char;   // Zellenkontrast (Wert) / Cell contrast (value)
      ccValue4 { ExternalAccessible := 'False'; ExternalVisible := 'False'; ExternalWritable := 'False'} : Char;   // Zellenkontrast (Wert) / Cell contrast (value)
      ccValue5 { ExternalAccessible := 'False'; ExternalVisible := 'False'; ExternalWritable := 'False'} : Char;   // Zellenkontrast (Wert) / Cell contrast (value)
      ccValue6 { ExternalAccessible := 'False'; ExternalVisible := 'False'; ExternalWritable := 'False'} : Char;   // Zellenkontrast (Wert) / Cell contrast (value)
      ccValue_comma { ExternalAccessible := 'False'; ExternalVisible := 'False'; ExternalWritable := 'False'} : Char := ',';   // Komma / Comma
      cm { ExternalAccessible := 'False'; ExternalVisible := 'False'; ExternalWritable := 'False'} : Char;   // Zellenmodulation / Cell modulation
      cm_comma { ExternalAccessible := 'False'; ExternalVisible := 'False'; ExternalWritable := 'False'} : Char := ',';   // Komma / Comma
      rm { ExternalAccessible := 'False'; ExternalVisible := 'False'; ExternalWritable := 'False'} : Char;   // Refelxtionsrand / Reflective edge
      rm_comma { ExternalAccessible := 'False'; ExternalVisible := 'False'; ExternalWritable := 'False'} : Char := ',';   // Komma / Comma
      fpd { ExternalAccessible := 'False'; ExternalVisible := 'False'; ExternalWritable := 'False'} : Char;   // Schäaden am festen Muster / Damage to the fixed sample
      fpd_comma { ExternalAccessible := 'False'; ExternalVisible := 'False'; ExternalWritable := 'False'} : Char := ',';   // Komma / Comma
      an { ExternalAccessible := 'False'; ExternalVisible := 'False'; ExternalWritable := 'False'} : Char;   // Axiale Verzerrung / Axial distortion
      an_comma { ExternalAccessible := 'False'; ExternalVisible := 'False'; ExternalWritable := 'False'} : Char := ',';   // Komma / Comma
      anValue1 { ExternalAccessible := 'False'; ExternalVisible := 'False'; ExternalWritable := 'False'} : Char;   // Axiale Verzerrung (Wert) / Axial distortion (value)
      anValue2 { ExternalAccessible := 'False'; ExternalVisible := 'False'; ExternalWritable := 'False'} : Char;   // Axiale Verzerrung (Wert) / Axial distortion (value)
      anValue3 { ExternalAccessible := 'False'; ExternalVisible := 'False'; ExternalWritable := 'False'} : Char;   // Axiale Verzerrung (Wert) / Axial distortion (value)
      anValue4 { ExternalAccessible := 'False'; ExternalVisible := 'False'; ExternalWritable := 'False'} : Char;   // Axiale Verzerrung (Wert) / Axial distortion (value)
      anValue5 { ExternalAccessible := 'False'; ExternalVisible := 'False'; ExternalWritable := 'False'} : Char;   // Axiale Verzerrung (Wert) / Axial distortion (value)
      anValue6 { ExternalAccessible := 'False'; ExternalVisible := 'False'; ExternalWritable := 'False'} : Char;   // Axiale Verzerrung (Wert) / Axial distortion (value)
      anValue_comma { ExternalAccessible := 'False'; ExternalVisible := 'False'; ExternalWritable := 'False'} : Char := ',';   // Komma / Comma
      gn { ExternalAccessible := 'False'; ExternalVisible := 'False'; ExternalWritable := 'False'} : Char;   // Rasterverzerrung / Grid distortion
      gn_comma { ExternalAccessible := 'False'; ExternalVisible := 'False'; ExternalWritable := 'False'} : Char := ',';   // Komma / Comma
      gnValue1 { ExternalAccessible := 'False'; ExternalVisible := 'False'; ExternalWritable := 'False'} : Char;   // Rasterverzerrung (Wert) / Grid distortion (value)
      gnValue2 { ExternalAccessible := 'False'; ExternalVisible := 'False'; ExternalWritable := 'False'} : Char;   // Rasterverzerrung (Wert) / Grid distortion (value)
      gnValue3 { ExternalAccessible := 'False'; ExternalVisible := 'False'; ExternalWritable := 'False'} : Char;   // Rasterverzerrung (Wert) / Grid distortion (value)
      gnValue4 { ExternalAccessible := 'False'; ExternalVisible := 'False'; ExternalWritable := 'False'} : Char;   // Rasterverzerrung (Wert) / Grid distortion (value)
      gnValue5 { ExternalAccessible := 'False'; ExternalVisible := 'False'; ExternalWritable := 'False'} : Char;   // Rasterverzerrung (Wert) / Grid distortion (value)
      gnValue6 { ExternalAccessible := 'False'; ExternalVisible := 'False'; ExternalWritable := 'False'} : Char;   // Rasterverzerrung (Wert) / Grid distortion (value)
      gnValue_comma { ExternalAccessible := 'False'; ExternalVisible := 'False'; ExternalWritable := 'False'} : Char := ',';   // Komma / Comma
      uec { ExternalAccessible := 'False'; ExternalVisible := 'False'; ExternalWritable := 'False'} : Char;   // Nicht verwendete Fehlerkorrektur / Unused error correction
      uec_comma { ExternalAccessible := 'False'; ExternalVisible := 'False'; ExternalWritable := 'False'} : Char := ',';   // Komma / Comma
      uecValue1 { ExternalAccessible := 'False'; ExternalVisible := 'False'; ExternalWritable := 'False'} : Char;   // Nicht verwendete Fehlerkorrektur (Wert) / Unused error correction (value)
      uecValue2 { ExternalAccessible := 'False'; ExternalVisible := 'False'; ExternalWritable := 'False'} : Char;   // Nicht verwendete Fehlerkorrektur (Wert) / Unused error correction (value)
      uecValue3 { ExternalAccessible := 'False'; ExternalVisible := 'False'; ExternalWritable := 'False'} : Char;   // Nicht verwendete Fehlerkorrektur (Wert) / Unused error correction (value)
      uecValue4 { ExternalAccessible := 'False'; ExternalVisible := 'False'; ExternalWritable := 'False'} : Char;   // Nicht verwendete Fehlerkorrektur (Wert) / Unused error correction (value)
      uecValue5 { ExternalAccessible := 'False'; ExternalVisible := 'False'; ExternalWritable := 'False'} : Char;   // Nicht verwendete Fehlerkorrektur (Wert) / Unused error correction (value)
      uecValue6 { ExternalAccessible := 'False'; ExternalVisible := 'False'; ExternalWritable := 'False'} : Char;   // Nicht verwendete Fehlerkorrektur (Wert) / Unused error correction (value)
      uecValue_comma { ExternalAccessible := 'False'; ExternalVisible := 'False'; ExternalWritable := 'False'} : Char := ',';   // Komma / Comma
      fid { ExternalAccessible := 'False'; ExternalVisible := 'False'; ExternalWritable := 'False'} : Char;   // Schaden an Formatdaten / Damage to format data
      fid_comma { ExternalAccessible := 'False'; ExternalVisible := 'False'; ExternalWritable := 'False'} : Char := ',';   // Komma / Comma
      fidValue1 { ExternalAccessible := 'False'; ExternalVisible := 'False'; ExternalWritable := 'False'} : Char;   // Schaden an Formatdaten (Wert) / Damage to format data (value)
      fidValue2 { ExternalAccessible := 'False'; ExternalVisible := 'False'; ExternalWritable := 'False'} : Char;   // Schaden an Formatdaten (Wert) / Damage to format data (value)
      fidValue3 { ExternalAccessible := 'False'; ExternalVisible := 'False'; ExternalWritable := 'False'} : Char;   // Schaden an Formatdaten (Wert) / Damage to format data (value)
      fidValue4 { ExternalAccessible := 'False'; ExternalVisible := 'False'; ExternalWritable := 'False'} : Char;   // Schaden an Formatdaten (Wert) / Damage to format data (value)
      fidValue5 { ExternalAccessible := 'False'; ExternalVisible := 'False'; ExternalWritable := 'False'} : Char;   // Schaden an Formatdaten (Wert) / Damage to format data (value)
      fidValue6 { ExternalAccessible := 'False'; ExternalVisible := 'False'; ExternalWritable := 'False'} : Char;   // Schaden an Formatdaten (Wert) / Damage to format data (value)
      fidValue_comma { ExternalAccessible := 'False'; ExternalVisible := 'False'; ExternalWritable := 'False'} : Char := ',';   // Komma / Comma
      vid { ExternalAccessible := 'False'; ExternalVisible := 'False'; ExternalWritable := 'False'} : Char;   // Modelldatenschaden / Model data damage
      vid_comma { ExternalAccessible := 'False'; ExternalVisible := 'False'; ExternalWritable := 'False'} : Char := ',';   // Komma / Comma
      vidValue1 { ExternalAccessible := 'False'; ExternalVisible := 'False'; ExternalWritable := 'False'} : Char;   // Modelldatenschaden (Wert) / Model data damage (value)
      vidValue2 { ExternalAccessible := 'False'; ExternalVisible := 'False'; ExternalWritable := 'False'} : Char;   // Modelldatenschaden (Wert) / Model data damage (value)
      vidValue3 { ExternalAccessible := 'False'; ExternalVisible := 'False'; ExternalWritable := 'False'} : Char;   // Modelldatenschaden (Wert) / Model data damage (value)
      vidValue4 { ExternalAccessible := 'False'; ExternalVisible := 'False'; ExternalWritable := 'False'} : Char;   // Modelldatenschaden (Wert) / Model data damage (value)
      vidValue5 { ExternalAccessible := 'False'; ExternalVisible := 'False'; ExternalWritable := 'False'} : Char;   // Modelldatenschaden (Wert) / Model data damage (value)
      vidValue6 { ExternalAccessible := 'False'; ExternalVisible := 'False'; ExternalWritable := 'False'} : Char;   // Modelldatenschaden (Wert) / Model data damage (value)
      vidValue_comma { ExternalAccessible := 'False'; ExternalVisible := 'False'; ExternalWritable := 'False'} : Char := ',';   // Komma / Comma
      pgh { ExternalAccessible := 'False'; ExternalVisible := 'False'; ExternalWritable := 'False'} : Char;   // Druckskalierung horizontal / Print scaling horizontal
      pgh_comma { ExternalAccessible := 'False'; ExternalVisible := 'False'; ExternalWritable := 'False'} : Char := ',';   // Komma / Comma
      pghValue1 { ExternalAccessible := 'False'; ExternalVisible := 'False'; ExternalWritable := 'False'} : Char;   // Druckskalierung horizontal (Wert) / Print scaling horizontal (value)
      pghValue2 { ExternalAccessible := 'False'; ExternalVisible := 'False'; ExternalWritable := 'False'} : Char;   // Druckskalierung horizontal (Wert) / Print scaling horizontal (value)
      pghValue3 { ExternalAccessible := 'False'; ExternalVisible := 'False'; ExternalWritable := 'False'} : Char;   // Druckskalierung horizontal (Wert) / Print scaling horizontal (value)
      pghValue4 { ExternalAccessible := 'False'; ExternalVisible := 'False'; ExternalWritable := 'False'} : Char;   // Druckskalierung horizontal (Wert) / Print scaling horizontal (value)
      pghValue5 { ExternalAccessible := 'False'; ExternalVisible := 'False'; ExternalWritable := 'False'} : Char;   // Druckskalierung horizontal (Wert) / Print scaling horizontal (value)
      pghValue6 { ExternalAccessible := 'False'; ExternalVisible := 'False'; ExternalWritable := 'False'} : Char;   // Druckskalierung horizontal (Wert) / Print scaling horizontal (value)
      pghValue_comma { ExternalAccessible := 'False'; ExternalVisible := 'False'; ExternalWritable := 'False'} : Char := ',';   // Komma / Comma
      pgv { ExternalAccessible := 'False'; ExternalVisible := 'False'; ExternalWritable := 'False'} : Char;   // Druckskalierung vertikal / Print scaling vertical
      pgv_comma { ExternalAccessible := 'False'; ExternalVisible := 'False'; ExternalWritable := 'False'} : Char := ',';   // Komma / Comma
      pgvValue1 { ExternalAccessible := 'False'; ExternalVisible := 'False'; ExternalWritable := 'False'} : Char;   // Druckskalierung vertikal (Wert) / Print scaling vertical (value)
      pgvValue2 { ExternalAccessible := 'False'; ExternalVisible := 'False'; ExternalWritable := 'False'} : Char;   // Druckskalierung vertikal (Wert) / Print scaling vertical (value)
      pgvValue3 { ExternalAccessible := 'False'; ExternalVisible := 'False'; ExternalWritable := 'False'} : Char;   // Druckskalierung vertikal (Wert) / Print scaling vertical (value)
      pgvValue4 { ExternalAccessible := 'False'; ExternalVisible := 'False'; ExternalWritable := 'False'} : Char;   // Druckskalierung vertikal (Wert) / Print scaling vertical (value)
      pgvValue5 { ExternalAccessible := 'False'; ExternalVisible := 'False'; ExternalWritable := 'False'} : Char;   // Druckskalierung vertikal (Wert) / Print scaling vertical (value)
      pgvValue6 { ExternalAccessible := 'False'; ExternalVisible := 'False'; ExternalWritable := 'False'} : Char;   // Druckskalierung vertikal (Wert) / Print scaling vertical (value)
      pgvValue_comma { ExternalAccessible := 'False'; ExternalVisible := 'False'; ExternalWritable := 'False'} : Char := ',';   // Komma / Comma
   END_STRUCT;
END_TYPE

TYPE "typeKeyenceHmi"
// V01.00
// stored: IsFailsafeCompliant false
   STRUCT
      Input : Struct   // Data from HMI
         StartLaser : Bool;   // Start Markiervorgang / Start marking process
         StartDmcRenew : Bool;   // Start DMC erneuern / Start renewing DMC
         ResetLaser : Bool;   // Reset Laser / Reset laser
         ResetFinishState : Bool;   // Fertigmeldung zurücksetzen / Finished message reset
         MistCollectorTrigger : Bool;   // Absaugung triggern / Trigger exhaust system / Trigger exhaust
         TeachDistanceSensor : Bool;   // Abstandsensor teachen / Teach distance sensor
         CameraTrigger : Bool;   // Kamera triggern / Trigger camera
         OffsetDistSensorDistance : Real;   // Offsetwert zum Abnullen des Abstandsensors / Offset value for resetting the distance sensor
         OffsetDistSensorAngle : Real;   // Offsetwert zum Abnullen des Abstandsensors / Offset value for resetting the distance sensor
      END_STRUCT;
      Output : Struct   // Data to HMI
         ElementVisible : Struct
            ButtonStartLaser : Bool;
            ButtonStartRenew : Bool;
            ButtonReset : Bool;
            ButtonResetFinishState : Bool;
            ButtonTrigMistCollector : Bool;
            ButtonTeachDistanceSensor : Bool;
            ButtonTriggerCamera : Bool;
            LabelStringData : Bool;
            LabelDmc : Bool;
            LabelPrgNr : Bool;
            LabelErrorCode : Bool;
            LabelFocus : Bool;
            LabelDistance : Bool;
            LabelMarkingTime : Bool;
            TextboxDistanceOffset : Bool;
            ImageMistCollector : Bool;
            ImageReadResult : Bool;
         END_STRUCT;
         ElementEnable : Struct
            ButtonStartLaser : Bool;
            ButtonStartRenew : Bool;
            ButtonReset : Bool;
            ButtonResetFinishState : Bool;
            ButtonTrigMistCollector : Bool;
            ButtonTeachDistanceSensor : Bool;
            TextboxDistanceOffset : Bool;
         END_STRUCT;
         ElementActive : Struct
            ButtonStartLaser : Bool;
            ButtonStartRenew : Bool;
            ButtonReset : Bool;
            ButtonResetFinishState : Bool;
            ButtonTrigMistCollector : Bool;
            ButtonTeachDistanceSensor : Bool;
         END_STRUCT;
         Data : Struct
            Image : Struct   // Steuerung HMI Bilder / Control HMI screens
               LaserReady : Byte;   // Laser Betriebsbereit / Laser ready for operation
               LaserSelected : Byte;   // Markiereinheit aktiv / Marking unit active
               WorkpieceInPosition : Byte;   // Werstkück in Position / Part in position
               SafetyCircuit : Byte;   // Schutzkreis / Protective circuit
               Error : Byte;   // Störung / Fault / Failure
               KeySwitch : Byte;   // Schlüsselschalter / Key-operated switch
               MistCollector : Byte;   // Absaugung / Exhaust system / Exhaust
               Laser : Byte;   // Laser
               Shutter : Byte;   // Verschluss / Seal
               LaserFinished : Byte;   // Fertigmeldung Laser / Finished message laser
               StartMarking : Byte;   // Start Markieren / Start marking
               StartRenew : Byte;   // Start DMC Renew / Start DMC renew
               ResetLaser : Byte;   // Reset Laser / Reset laser
               quality : Byte;   // Leseergebnis / Qualität / Reset laser / Read result/quality
            END_STRUCT;
            LaserStatus : Struct
               TriggerReady : Bool;
               Error : Bool;
               Warning : Bool;
               Notice : Bool;
               Shutter : Bool;
               StartUp : Bool;
               res_0_6 : Bool;
               res_0_7 : Bool;
               Laser_Emit : Bool;
               ShutterControl : Bool;
               RemoteInterlock : Bool;
               Contacter : Bool;
               res_1_4 : Bool;
               res_1_5 : Bool;
               res_1_6 : Bool;
               res_1_7 : Bool;
               Busy : Bool;
               PrintBusy : Bool;
               GuidePrintBusy : Bool;
               ChangeBusy : Bool;
               LockBusy : Bool;
               EditBusy : Bool;
               Code2DReaderBusy : Bool;
               res_2_7 : Bool;
               res_3_0 : Bool;
               res_3_1 : Bool;
               res_3_2 : Bool;
               res_3_3 : Bool;
               res_3_4 : Bool;
               res_3_5 : Bool;
               res_3_6 : Bool;
               res_3_7 : Bool;
            END_STRUCT;
            ErrorCodeIntern : Int;   // interner Fehler Code / RESPONSE - VALUE 1 / Internal error code
            CharacterString : String[100];   // DMC Beschriftungsinhalt / DMC labeling content
            ReadDmc : String;   // gelesener DMC / Read DMC
            Status : Byte;   // aktueller Status / Current status
            CommandActive : Bool;   // Ablauf aktiv / Sequence active
            Offset : Struct   // Anzeige der hinterlegten Parameter Offsets / Display of stored parameter offsets
               Power : Real;   // aktueller Offset: Leistung / Current offset: power
               Frequence : Real;   // aktueller Offset: Frequenz / Current offset: frequency
               Speed : Real;   // aktueller Offset: Geschwindigkeit / Current offset: speed
               Defocus : Real;   // aktueller Offset: Defokus / Current offset: defocus
               Pulse_Width : Real;   // aktueller Offset: Pulsweite / Current offset: pulse width
            END_STRUCT;
            DistanceSensor : Struct   // Anzeige Abstandsensor / Display distance sensor
               Difference : Real;   // Differenz: Settingwert - Aktualwert / Difference: setting value - current value
               CurrentValue : Real;   // Aktualwert / Current value
               SettingValue : Real;   // Settingwert / Setting value
               Offset : Real;
            END_STRUCT;
            Zusatinformationen : Struct
               PrgNr : Array[1..4] of Char;   // Programmnummer / Loaded marking file / Program number
               ErrorCodesLaser : Array[1..3] of Int;   // Fehler Codes vom Laser / Error codes from the laser
               CommandError : Word;
               MarkingTime : Real;   // Beschriftungszeit - Markiervorgang / Labeling time - marking process
               TotalTime : Real;   // Beschriftungszeit - Gesamtablauf / Labeling time - complete cycle
               Length : Int;
               DataMatrix : Array[1..100] of Char;
            END_STRUCT;
         END_STRUCT;
      END_STRUCT;
   END_STRUCT;
END_TYPE

TYPE "typeMotionOvrvList"
TITLE = Motion overview list / Motion-Übersichtsliste
// Motion overview list [V 01.00 | Kernel_V2] / Motion-Übersichtsliste [V 01.00 | Kernel_V2]
// stored: IsFailsafeCompliant false
   STRUCT
      enabled : Bool;   // Motion-Übersicht ist freigeschaltet / Motion overview is activated
      lastUsedIndex : DInt := -1;   // Letzter Benutzter Index / Last user index
      valid : Bool;   // Gültigkeit / Scope
      overflowCount : DInt;   // Gruppen Überlauf Zähler / Groups overtravel counter
      motions : Array[0.."MAX_CNT_MTN_OVR_ENTRIES"] of "typeMotionOvrvListEntry";   // Motions
   END_STRUCT;
END_TYPE

TYPE "typeMotionOvrvListEntry"
TITLE = Entry motion overview / Eintrag Motion-Übersicht
// Entry motion overview [V 01.00 | Kernel_V2] / Eintrag Motion-Übersicht [V 01.00 | Kernel_V2]
// stored: IsFailsafeCompliant false
   STRUCT
      alive : USInt;   // Alive-Flag (Wird im Motion gesetzt, zentral dann zurückgesetzt) / Alive-Flag (is set in motion, then centrally reset)
      instancePath : String[80];   // Instanzpfad des Motion-Aufrufes (Dient als Identifier) / Instance path of motion call (serves as identifier)
      fgDbAdress : DB_ANY;   // DB-Any Adresse der zugehörigen Funktionsgruppe / DB any address of associated function group
      data : Struct   // Motion-Daten:... / Motion data...
         enable : Bool;   // Grundsätzliche Freigabesignale (Steuerung ein, usw.) / Basic enabling signals (control system on, etc.)
         interlock : Bool;   // Bewegungsverriegelung / Motion interlock
         toPosition : Bool;   // Zur Position aktiv / To position active
         inPosition : Bool;   // In Position / In position
         inPositionStored : Bool;   // Position wurde in Automatik angefahren und wird überwacht / Position was approached in automatic mode and is monitored
         positionValue : LReal;   // Positionswert (optional) / Position value (optional)
         timeOut : Time;   // Überwachungszeit für die Bewegung / Monitoring time for the motion
         timeOfLastMotion : Time;   // Tatsächlich benötigte Zeit der letzten Bewegung / Actually required time of the last motion
      END_STRUCT;
      hmiLine : Struct   // HMI-Zeileninformation / HMI line information
         number : UInt;   // Zeilennummer (0 = keine Zeile) / Line number (0 = no line)
         controSide : SInt;   // Einrichtzeile Links/Rechts (-1 = Links, 0 = keine, 1 = Rechts) / Setup line left/right (-1 = left, 0 = none, 1 = right)
      END_STRUCT;
   END_STRUCT;
END_TYPE

DATA_BLOCK "Dummy_LaserComm"   // DB6
{ S7_Optimized_Access := 'TRUE' }
VERSION : 0.1
// stored: AutoNumber true, DBAccessibleFromOPCUA true, DBAccessibleFromWebserver true, IsOnlyStoredInLoadMemory false, IsRetainMemResEnabled false, IsWriteProtectedInAS false, MemoryReserve 100
   VAR
      iScanner : "Scanner_Inputs";
      oScanner { S7_SetPoint := 'True'} : "Scanner_Outputs";
      iSource { S7_SetPoint := 'True'} : "YLS_Inputs";
      oSource : "YLS_Outputs";
   END_VAR
BEGIN
END_DATA_BLOCK

DATA_BLOCK "FgLaser1Control"   // DB180
TITLE = FG $[name] Control system / FG $[name] Steuerung
{ S7_Optimized_Access := 'TRUE'; DB_Accessible_From_OPC_UA := 'FALSE' }
FAMILY : FG
VERSION : 0.0.0.0
// FG $[name] Control system / FG $[name] Steuerung
// stored: AutoNumber true, DBAccessibleFromOPCUA false, DBAccessibleFromWebserver true, IsOnlyStoredInLoadMemory false, IsRetainMemResEnabled false, IsWriteProtectedInAS false, MemoryReserve 100
   VAR
      general { ExternalAccessible := 'False'; ExternalVisible := 'False'; ExternalWritable := 'False'} : "typeFgControlGeneral";   // FG Laser 1: Allgemein / FG Laser 1: general
      activeJob { ExternalAccessible := 'False'; ExternalVisible := 'False'; ExternalWritable := 'False'} : Struct   // FG Laser 1: Aktiver Auftrag / FG Laser 1: active job
         job1SealAirOn { ExternalAccessible := 'False'; ExternalVisible := 'False'; ExternalWritable := 'False'} : Bool;   // FG Laser 1 - Auftrag 1: Sperrluft einschalten aktiv / FG Laser 1 - job 1: switch on sealing air active
         job2LaserOn { ExternalAccessible := 'False'; ExternalVisible := 'False'; ExternalWritable := 'False'} : Bool;   // FG Laser 1 - Auftrag 2: Laser ein aktiv / FG Laser 1 - job 2: laser on active
         job3SealAirOff { ExternalAccessible := 'False'; ExternalVisible := 'False'; ExternalWritable := 'False'} : Bool;   // FG Laser 1 - Auftrag 3: Sperrluft ausschalten aktiv / FG Laser 1 - job 3: switch off sealing air active
         job4LaserOnSpecialFunction { ExternalAccessible := 'False'; ExternalVisible := 'False'; ExternalWritable := 'False'} : Bool;   // FG Laser 1 - Auftrag 4: Laser ein Sonderablauf aktiv / FG Laser 1 - job 4: laser on special sequence active
         job99ToHomePos { ExternalAccessible := 'False'; ExternalVisible := 'False'; ExternalWritable := 'False'} : Bool;   // FG Laser 1 - Auftrag 99: Zur Grundstellung aktiv / FG Laser 1 - Job 99: To home position active
      END_STRUCT;
      motions { ExternalAccessible := 'False'; ExternalVisible := 'False'; ExternalWritable := 'False'} : Struct   // FG Laser 1: Bewegungen / FG laser 1: Motions
         switchOnSealAir { ExternalAccessible := 'False'; ExternalVisible := 'False'; ExternalWritable := 'False'} : "typeMotion";   // FG Laser 1: Sperrluft einschalten / FG Laser 1: Switch on sealing air
         switchOffSealAir { ExternalAccessible := 'False'; ExternalVisible := 'False'; ExternalWritable := 'False'} : "typeMotion";   // FG Laser 1: Sperrluft ausschalten / FG Laser 1: Switch off sealing air
         switchOnProtectionGas1_1 { ExternalAccessible := 'False'; ExternalVisible := 'False'; ExternalWritable := 'False'} : "typeMotion";   // FG Laser 1: Schutzgas 1.1 einschalten / FG laser 1: Switch on shielding gas 1.1
         switchOffProtectionGas1_1 { ExternalAccessible := 'False'; ExternalVisible := 'False'; ExternalWritable := 'False'} : "typeMotion";   // FG Laser 1: Schutzgas 1.1 ausschalten / FG laser 1: Switch off shielding gas 1.1
         switchOnProtectionGas1_2 { ExternalAccessible := 'False'; ExternalVisible := 'False'; ExternalWritable := 'False'} : "typeMotion";   // FG Laser 1: Schutzgas 1.2 einschalten / FG laser 1: Switch on shielding gas 1.2
         switchOffProtectionGas1_2 { ExternalAccessible := 'False'; ExternalVisible := 'False'; ExternalWritable := 'False'} : "typeMotion";   // FG Laser 1: Schutzgas 1.2 ausschalten / FG laser 1: Switch off shielding gas 1.2
         switchOnProtectionGas1_3 { ExternalAccessible := 'False'; ExternalVisible := 'False'; ExternalWritable := 'False'} : "typeMotion";   // FG Laser 1: Schutzgas 1.3 einschalten / FG laser 1: Switch on shielding gas 1.3
         switchOffProtectionGas1_3 { ExternalAccessible := 'False'; ExternalVisible := 'False'; ExternalWritable := 'False'} : "typeMotion";   // FG Laser 1: Schutzgas 1.3 ausschalten / FG laser 1: Switch off shielding gas 1.3
         switchOnProtectionGas1_4 { ExternalAccessible := 'False'; ExternalVisible := 'False'; ExternalWritable := 'False'} : "typeMotion";   // FG Laser 1: Schutzgas 1.4 einschalten / FG laser 1: Switch on shielding gas 1.4
         switchOffProtectionGas1_4 { ExternalAccessible := 'False'; ExternalVisible := 'False'; ExternalWritable := 'False'} : "typeMotion";   // FG Laser 1: Schutzgas 1.4 ausschalten / FG laser 1: Switch off shielding gas 1.4
         switchOnProtectionGas1_5 { ExternalAccessible := 'False'; ExternalVisible := 'False'; ExternalWritable := 'False'} : "typeMotion";   // FG Laser 1: Schutzgas 1.5 einschalten / FG laser 1: Switch on shielding gas 1.5
         switchOffProtectionGas1_5 { ExternalAccessible := 'False'; ExternalVisible := 'False'; ExternalWritable := 'False'} : "typeMotion";   // FG Laser 1: Schutzgas 1.5 ausschalten / FG laser 1: Switch off shielding gas 1.5
         switchOnProtectionGas1_6 { ExternalAccessible := 'False'; ExternalVisible := 'False'; ExternalWritable := 'False'} : "typeMotion";   // FG Laser 1: Schutzgas 1.6 einschalten / FG laser 1: Switch on shielding gas 1.6
         switchOffProtectionGas1_6 { ExternalAccessible := 'False'; ExternalVisible := 'False'; ExternalWritable := 'False'} : "typeMotion";   // FG Laser 1: Schutzgas 1.6 ausschalten / FG laser 1: Switch off shielding gas 1.6
         switchOnProtectionGasCalibration { ExternalAccessible := 'False'; ExternalVisible := 'False'; ExternalWritable := 'False'} : "typeMotion";   // FG Laser 1: Schutzgas Kalibriersystem einschalten / FG laser 1: Switch on shielding gas calibration system
         switchOffProtectionGasComplete { ExternalAccessible := 'False'; ExternalVisible := 'False'; ExternalWritable := 'False'} : "typeMotion";   // FG Laser 1: Schutzgas Laser 1 komplett ausschalten
         switchOffProtectionGasCalibration { ExternalAccessible := 'False'; ExternalVisible := 'False'; ExternalWritable := 'False'} : "typeMotion";   // FG Laser 1: Schutzgas Kalibriersystem ausschalten / FG laser 1: Switch off shielding gas calibration system
      END_STRUCT;
      laserTaskCurrent { ExternalAccessible := 'False'; ExternalVisible := 'False'; ExternalWritable := 'False'} : Bool;   // FG Laser 1: Laser Task Aktiv / FG Laser 1: Laser task active
      laserEvaluationNotActive { ExternalAccessible := 'False'; ExternalVisible := 'False'; ExternalWritable := 'False'} : Bool;   // FG Laser 1: Laser Auswertung nicht aktiv / FG Laser 1: Laser evaluation not active
   END_VAR
   VAR RETAIN
      laserMeasuring { ExternalAccessible := 'False'; ExternalVisible := 'False'; ExternalWritable := 'False'} : Struct   // FG Laser 1: Lasermessungen / FG laser 1: Laser measurements
         powerMeasuringRequest { ExternalAccessible := 'False'; ExternalVisible := 'False'; ExternalWritable := 'False'} : Bool;   // FG Laser 1: Laserleistungsmessung Anforderung / FG laser 1: laser power measurement request
         powerMeasuringStart { ExternalAccessible := 'False'; ExternalVisible := 'False'; ExternalWritable := 'False'} : Bool;   // FG Laser 1: Laserleistungsmessung starten / FG laser 1: Start laser power measurement
         powerMeasuringDone { ExternalAccessible := 'False'; ExternalVisible := 'False'; ExternalWritable := 'False'} : Bool;   // FG Laser 1: Laserleistungsmessung beendet / FG laser 1: laser power measurement not completed
         beamWatchMeasuringRequest { ExternalAccessible := 'False'; ExternalVisible := 'False'; ExternalWritable := 'False'} : Bool;   // FG Laser 1: BeamWatchmessung Anforderung / FG laser 1: BeamWatchmeasurement request
         beamWatchMeasuringStart { ExternalAccessible := 'False'; ExternalVisible := 'False'; ExternalWritable := 'False'} : Bool;   // FG Laser 1: BeamWatchmessung starten / FG Laser 1: Start Beamwatch measurement
         beamWatchMeasuringDone { ExternalAccessible := 'False'; ExternalVisible := 'False'; ExternalWritable := 'False'} : Bool;   // FG Laser 1: BeamWatchmessung beendet / FG laser 1: BeamWatchmeasurement not finished
         lddCalibrationRequest { ExternalAccessible := 'False'; ExternalVisible := 'False'; ExternalWritable := 'False'} : Bool;   // FG Laser 1: LDD Kalibrierung Anforderung / FG laser 1: LDD calibration request
         lddCalibrationStart { ExternalAccessible := 'False'; ExternalVisible := 'False'; ExternalWritable := 'False'} : Bool;   // FG Laser 1: LDD Kalibrierung starten / FG laser 1: start LDD calibration
         lddCalibrationDone { ExternalAccessible := 'False'; ExternalVisible := 'False'; ExternalWritable := 'False'} : Bool;   // FG Laser 1: LDD Kalibrierung beendet / FG laser 1: LDD calibration not finished
         changeCalibrationPieceDone { ExternalAccessible := 'False'; ExternalVisible := 'False'; ExternalWritable := 'False'} : Bool;   // FG Laser 1: Opferblech LDD Kalibrierung tauschen beendet / FG laser 1: Change sacrificial part LDD calibration finished
         ready { ExternalAccessible := 'False'; ExternalVisible := 'False'; ExternalWritable := 'False'} : Bool;   // FG Laser 1: Lasermessung bereit / FG laser 1: Laser measurement ready
      END_STRUCT;
   END_VAR
   VAR
      dryRunWeldSimDone { ExternalAccessible := 'False'; ExternalVisible := 'False'; ExternalWritable := 'False'} : Bool;   // FG Laser 1: Trockenlauf der Schweißsimulation durchgeführt / FG laser 1: dry run of welding simulation performed
      dryRunWeldSimOk { ExternalAccessible := 'False'; ExternalVisible := 'False'; ExternalWritable := 'False'} : Bool := TRUE;   // FG Laser 1: Ergebnis der Trockenschweißung: Aufgabe einstellen OK / FG laser 1: result of dry welding: set task OK
      SMCstatus { ExternalAccessible := 'False'; ExternalVisible := 'False'; ExternalWritable := 'False'} : "typeSmcChillerHrle90a40cmStatus";   // FG Laser 1: SMC Kühler / FG Laser 1: SMC cooler
      laserManOnBypassEnable { ExternalAccessible := 'False'; ExternalVisible := 'False'; ExternalWritable := 'False'} : Bool;   // FG Laser 1: Aktiviert die Umgehung einiger Regeln, um den Laser einzuschalten / FG Laser 1: Activates the bypass of some rules to switch on the laser
   END_VAR
   VAR RETAIN
      analogSensor { ExternalAccessible := 'False'; ExternalVisible := 'False'; ExternalWritable := 'False'} : Struct   // FG Laser 1: Analogsensoren
         FlowProtGas1_1 { ExternalAccessible := 'False'; ExternalVisible := 'False'; ExternalWritable := 'False'} : Struct   // FG Laser 1: Durchflusssensor Schutzgas 1.1
            limitsSensor { ExternalAccessible := 'False'; ExternalVisible := 'False'; ExternalWritable := 'False'} : "typeAnalogSensorUniversalLimits";   // FG Laser 1: Durchflusssensor Schutzgas 1.1 Limits
            positionsSensor { ExternalAccessible := 'False'; ExternalVisible := 'False'; ExternalWritable := 'False'} : "typeAnalogSensorUniversalPositions";   // FG Laser 1: Durchflusssensor Schutzgas 1.1 Positionen
         END_STRUCT;
         FlowProtGas1_2 { ExternalAccessible := 'False'; ExternalVisible := 'False'; ExternalWritable := 'False'} : Struct   // FG Laser 1: Durchflusssensor Schutzgas 1.2
            limitsSensor { ExternalAccessible := 'False'; ExternalVisible := 'False'; ExternalWritable := 'False'} : "typeAnalogSensorUniversalLimits";   // FG Laser 1: Durchflusssensor Schutzgas 1.2 Limits
            positionsSensor { ExternalAccessible := 'False'; ExternalVisible := 'False'; ExternalWritable := 'False'} : "typeAnalogSensorUniversalPositions";   // FG Laser 1: Durchflusssensor Schutzgas 1.2 Positionen
         END_STRUCT;
         FlowProtGas1_3 { ExternalAccessible := 'False'; ExternalVisible := 'False'; ExternalWritable := 'False'} : Struct   // FG Laser 1: Durchflusssensor Schutzgas 1.3
            limitsSensor { ExternalAccessible := 'False'; ExternalVisible := 'False'; ExternalWritable := 'False'} : "typeAnalogSensorUniversalLimits";   // FG Laser 1: Durchflusssensor Schutzgas 1.3 Limits
            positionsSensor { ExternalAccessible := 'False'; ExternalVisible := 'False'; ExternalWritable := 'False'} : "typeAnalogSensorUniversalPositions";   // FG Laser 1: Durchflusssensor Schutzgas 1.3 Positionen
         END_STRUCT;
         FlowProtGas1_4 { ExternalAccessible := 'False'; ExternalVisible := 'False'; ExternalWritable := 'False'} : Struct   // FG Laser 1: Durchflusssensor Schutzgas 1.4
            limitsSensor { ExternalAccessible := 'False'; ExternalVisible := 'False'; ExternalWritable := 'False'} : "typeAnalogSensorUniversalLimits";   // FG Laser 1: Durchflusssensor Schutzgas 1.4 Limits
            positionsSensor { ExternalAccessible := 'False'; ExternalVisible := 'False'; ExternalWritable := 'False'} : "typeAnalogSensorUniversalPositions";   // FG Laser 1: Durchflusssensor Schutzgas 1.4 Positionen
         END_STRUCT;
         FlowProtGas1_5 { ExternalAccessible := 'False'; ExternalVisible := 'False'; ExternalWritable := 'False'} : Struct   // FG Laser 1: Durchflusssensor Schutzgas 1.5
            limitsSensor { ExternalAccessible := 'False'; ExternalVisible := 'False'; ExternalWritable := 'False'} : "typeAnalogSensorUniversalLimits";   // FG Laser 1: Durchflusssensor Schutzgas 1.5 Limits
            positionsSensor { ExternalAccessible := 'False'; ExternalVisible := 'False'; ExternalWritable := 'False'} : "typeAnalogSensorUniversalPositions";   // FG Laser 1: Durchflusssensor Schutzgas 1.5 Positionen
         END_STRUCT;
         FlowProtGas1_6 { ExternalAccessible := 'False'; ExternalVisible := 'False'; ExternalWritable := 'False'} : Struct   // FG Laser 1: Durchflusssensor Schutzgas 1.6
            limitsSensor { ExternalAccessible := 'False'; ExternalVisible := 'False'; ExternalWritable := 'False'} : "typeAnalogSensorUniversalLimits";   // FG Laser 1: Durchflusssensor Schutzgas 1.6 Limits
            positionsSensor { ExternalAccessible := 'False'; ExternalVisible := 'False'; ExternalWritable := 'False'} : "typeAnalogSensorUniversalPositions";   // FG Laser 1: Durchflusssensor Schutzgas 1.6 Positionen
         END_STRUCT;
      END_STRUCT;
   END_VAR
   VAR
      UsageCounterCalibrationPiece { ExternalAccessible := 'False'; ExternalVisible := 'False'; ExternalWritable := 'False'} : Struct   // FG Laser 1: Verschleisszähler Opferblech 1 / FG laser 1: wear counter sacrificial plate 1
         prewarning { ExternalAccessible := 'False'; ExternalVisible := 'False'; ExternalWritable := 'False'} : Bool;   // FG Laser 1: Vorwarnung des Zählers für Opferblech 1 / FG laser 1: prewarning of counter for sacrificial plate 1
         warning { ExternalAccessible := 'False'; ExternalVisible := 'False'; ExternalWritable := 'False'} : Bool;   // FG Laser 1: Warnung des Zählers für Opferblech 1 / FG laser 1: warning of counter for sacrificial plate 1
         error { ExternalAccessible := 'False'; ExternalVisible := 'False'; ExternalWritable := 'False'} : Bool;   // FG Laser 1: Zähler für Opferblech 1 erreicht / FG laser 1: counter for sacrificial plate 1 reached
      END_STRUCT;
      UsageCounterProtectionGlass { ExternalAccessible := 'False'; ExternalVisible := 'False'; ExternalWritable := 'False'} : Struct   // FG Laser 1: Verschleißzähler Schutglas / FG laser 1: wear counter protective glass
         prewarning { ExternalAccessible := 'False'; ExternalVisible := 'False'; ExternalWritable := 'False'} : Bool;   // FG Laser 1: Vorwarnung des Zählers für Schutzglas Laser 1 / FG laser 1: prewarning of counter for protective glass laser 1
         warning { ExternalAccessible := 'False'; ExternalVisible := 'False'; ExternalWritable := 'False'} : Bool;   // FG Laser 1: Warnung des Zählers für Schutglas Laser 1 / FG laser 1: warning of counter for protective glass laser 1
         error { ExternalAccessible := 'False'; ExternalVisible := 'False'; ExternalWritable := 'False'} : Bool;   // FG Laser 1: Zähler für Schutzglas erreicht Laser 1 / FG laser 1: counter for protective glass reached laser 1
      END_STRUCT;
      CalibrationPieceChanged { ExternalAccessible := 'False'; ExternalVisible := 'False'; ExternalWritable := 'False'} : Bool;   // FG Laser 1: Opferblech muss getauscht werden / FG laser 1: sacrificial plate must be replaced
   END_VAR
BEGIN
   // motions.switchOnSealAir.inPosition : FG Laser 1: Sperrluft eingeschalten / FG Laser 1: Sealing air switched on
   // motions.switchOnSealAir.autoInPos : FG Laser 1: Sperrluft eingeschalten (Automatic) / FG Laser 1: Sealing air switched on (automatic)
   // motions.switchOffSealAir.inPosition : FG Laser 1: Sperrluft ausgeschalten / FG Laser 1: Sealing air switched off
   // motions.switchOffSealAir.autoInPos : FG Laser 1: Sperrluft ausgeschalten (Automatic) / FG Laser 1: Sealing air switched off (automatic)
   // motions.switchOnProtectionGas1_1.inPosition : FG Laser 1: Schutzgas 1.1 eingeschalten / FG laser 1: Shielding gas 1.1 switched on
   // motions.switchOnProtectionGas1_1.autoInPos : FG Laser 1: Schutzgas 1.1 eingeschalten (Automatic) / FG laser 1: Shielding gas 1.1 switched on (automatic)
   // motions.switchOffProtectionGas1_1.inPosition : FG Laser 1: Schutzgas 1.1 ausgeschalten / FG laser 1: Shielding gas 1.1 switched off
   // motions.switchOffProtectionGas1_1.autoInPos : FG Laser 1: Schutzgas 1.1 ausgeschalten (Automatic) / FG laser 1: Shielding gas 1.1 switched off (automatic)
   // motions.switchOnProtectionGas1_2.inPosition : FG Laser 1: Schutzgas 1.2 eingeschalten / FG laser 1: Shielding gas 1.2 switched on
   // motions.switchOnProtectionGas1_2.autoInPos : FG Laser 1: Schutzgas 1.2 eingeschalten (Automatic) / FG laser 1: Shielding gas 1.2 switched on (automatic)
   // motions.switchOffProtectionGas1_2.inPosition : FG Laser 1: Schutzgas 1.2 ausgeschalten / FG laser 1: Shielding gas 1.2 switched off
   // motions.switchOffProtectionGas1_2.autoInPos : FG Laser 1: Schutzgas 1.2 ausgeschalten (Automatic) / FG laser 1: Shielding gas 1.2 switched off (automatic)
   // motions.switchOnProtectionGas1_3.inPosition : FG Laser 1: Schutzgas 1.3 eingeschalten / FG laser 1: Shielding gas 1.3 switched on
   // motions.switchOnProtectionGas1_3.autoInPos : FG Laser 1: Schutzgas 1.3 eingeschalten (Automatic) / FG laser 1: Shielding gas 1.3 switched on (automatic)
   // motions.switchOffProtectionGas1_3.inPosition : FG Laser 1: Schutzgas 1.3 ausgeschalten / FG laser 1: Shielding gas 1.3 switched off
   // motions.switchOffProtectionGas1_3.autoInPos : FG Laser 1: Schutzgas 1.3 ausgeschalten (Automatic) / FG laser 1: Shielding gas 1.3 switched off (automatic)
   // motions.switchOnProtectionGas1_4.inPosition : FG Laser 1: Schutzgas 1.4 eingeschalten / FG laser 1: Shielding gas 1.4 switched on
   // motions.switchOnProtectionGas1_4.autoInPos : FG Laser 1: Schutzgas 1.4 eingeschalten (Automatic) / FG laser 1: Shielding gas 1.4 switched on (automatic)
   // motions.switchOffProtectionGas1_4.inPosition : FG Laser 1: Schutzgas 1.4 ausgeschalten / FG laser 1: Shielding gas 1.4 switched off
   // motions.switchOffProtectionGas1_4.autoInPos : FG Laser 1: Schutzgas 1.4 ausgeschalten (Automatic) / FG laser 1: Shielding gas 1.4 switched off (automatic)
   // motions.switchOnProtectionGas1_5.inPosition : FG Laser 1: Schutzgas 1.5 eingeschalten / FG laser 1: Shielding gas 1.5 switched on
   // motions.switchOnProtectionGas1_5.autoInPos : FG Laser 1: Schutzgas 1.5 eingeschalten (Automatic) / FG laser 1: Shielding gas 1.5 switched on (automatic)
   // motions.switchOffProtectionGas1_5.inPosition : FG Laser 1: Schutzgas 1.5 ausgeschalten / FG laser 1: Shielding gas 1.5 switched off
   // motions.switchOffProtectionGas1_5.autoInPos : FG Laser 1: Schutzgas 1.5 ausgeschalten (Automatic) / FG laser 1: Shielding gas 1.5 switched off (automatic)
   // motions.switchOnProtectionGas1_6.inPosition : FG Laser 1: Schutzgas 1.6 eingeschalten / FG laser 1: Shielding gas 1.6 switched on
   // motions.switchOnProtectionGas1_6.autoInPos : FG Laser 1: Schutzgas 1.6 eingeschalten (Automatic) / FG laser 1: Shielding gas 1.6 switched on (automatic)
   // motions.switchOffProtectionGas1_6.inPosition : FG Laser 1: Schutzgas 1.6 ausgeschalten / FG laser 1: Shielding gas 1.6 switched off
   // motions.switchOffProtectionGas1_6.autoInPos : FG Laser 1: Schutzgas 1.6 ausgeschalten (Automatic) / FG laser 1: Shielding gas 1.6 switched off (automatic)
   // motions.switchOnProtectionGasCalibration.inPosition : FG Laser 1: Schutzgas Kalibriersystem eingeschalten / FG laser 1: Shielding gas calibration system switched on
   // motions.switchOnProtectionGasCalibration.autoInPos : FG Laser 1: Schutzgas Kalibriersystem eingeschalten (Automatic) / FG laser 1: Shielding gas calibration system switched on (automatic)
   // motions.switchOffProtectionGasComplete.inPosition : FG Laser 1: Schutzgas Kalibriersystem ausgeschalten / FG laser 1: Shielding gas calibration system switched off
   // motions.switchOffProtectionGasComplete.autoInPos : FG Laser 1: Schutzgas Kalibriersystem ausgeschalten (Automatic) / FG laser 1: Shielding gas calibration system switched off (automatic)
   // motions.switchOffProtectionGasCalibration.inPosition : FG Laser 1: Schutzgas Kalibriersystem ausgeschalten / FG laser 1: Shielding gas calibration system switched off
   // motions.switchOffProtectionGasCalibration.autoInPos : FG Laser 1: Schutzgas Kalibriersystem ausgeschalten (Automatic) / FG laser 1: Shielding gas calibration system switched off (automatic)
END_DATA_BLOCK

DATA_BLOCK "LaserComm"   // DB295
{ S7_Optimized_Access := 'FALSE' }
VERSION : 0.1
// stored: AutoNumber true, DBAccessibleFromOPCUA true, DBAccessibleFromWebserver true, IsOnlyStoredInLoadMemory false, IsWriteProtectedInAS false
   VAR RETAIN
      "Version" : DInt;
      LDD_Array_Size : DInt;
      Instance : Array[0.."LASERCOMM_NUMBER_OF_LASERS"] of "LaserComm_Instance";
      "this CU" : "typeCaCgFg";
      fg_ControlGeneral { S7_SetPoint := 'True'} : "typeFgControlGeneral";
   END_VAR
BEGIN
END_DATA_BLOCK

ORGANIZATION_BLOCK "Main"   // OB1, LAD, ProgramCycle
TITLE = "Main Program Sweep (Cycle)"
{ S7_Optimized_Access := 'TRUE' }
VERSION : 0.1
// stored: AutoNumber true, IsIECCheckEnabled false, SetENOAutomatically false
   VAR_INPUT
      Initial_Call : Bool;   // Initial call of this OB
      Remanence : Bool;   // =True, if remanent data are available
   END_VAR
   VAR_TEMP
      Ack_Fault : Bool;
   END_VAR
BEGIN

REGION Network 1: Test Weld Sequence Reset
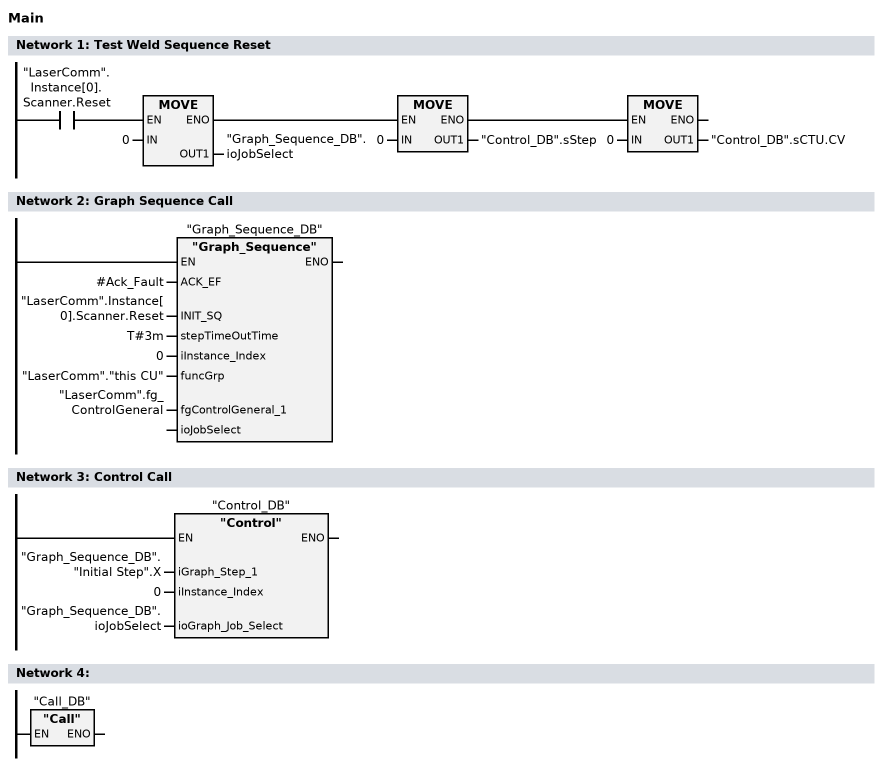
   RUNG wire#powerrail
      Contact( "LaserComm".Instance[0].Scanner.Reset )
      Move(in := 0, out1 => "Graph_Sequence_DB".ioJobSelect)
      Move(in := 0, out1 => "Control_DB".sStep)
      Move(in := 0, out1 => "Control_DB".sCTU.CV)
   END_RUNG
   // the same network as SCL:
   IF "LaserComm".Instance[0].Scanner.Reset THEN
       "Graph_Sequence_DB".ioJobSelect := 0;
       "Control_DB".sStep := 0;
       "Control_DB".sCTU.CV := 0;
   END_IF;
END_REGION

REGION Network 2: Graph Sequence Call
   RUNG wire#powerrail
      "Graph_Sequence_DB"(ACK_EF := #Ack_Fault, INIT_SQ := "LaserComm".Instance[0].Scanner.Reset, stepTimeOutTime := T#3m, iInstance_Index := 0, funcGrp := "LaserComm"."this CU", fgControlGeneral_1 := "LaserComm".fg_ControlGeneral, ioJobSelect :=)
   END_RUNG
   // the same network as SCL:
   "Graph_Sequence_DB"(ACK_EF := #Ack_Fault,   // "Graph_Sequence"
                       INIT_SQ := "LaserComm".Instance[0].Scanner.Reset,
                       stepTimeOutTime := T#3m,
                       iInstance_Index := 0,
                       funcGrp := "LaserComm"."this CU",
                       fgControlGeneral_1 := "LaserComm".fg_ControlGeneral);
END_REGION

REGION Network 3: Control Call
   RUNG wire#powerrail
      "Control_DB"(iGraph_Step_1 := "Graph_Sequence_DB"."Initial Step".X, iInstance_Index := 0, ioGraph_Job_Select := "Graph_Sequence_DB".ioJobSelect)
   END_RUNG
   // the same network as SCL:
   "Control_DB"(iGraph_Step_1 := "Graph_Sequence_DB"."Initial Step".X,   // "Control"
                iInstance_Index := 0,
                ioGraph_Job_Select := "Graph_Sequence_DB".ioJobSelect);
END_REGION

REGION Network 4
   RUNG wire#powerrail
      "Call_DB"()
   END_RUNG
   // the same network as SCL:
   "Call_DB"();   // "Call"
END_REGION
END_ORGANIZATION_BLOCK

